LIN {X 0,Y 336.702,Z 407.414,A -85,B 0,C 180,E1 14263.606,E2 14263.606} C_VEL
LIN {X 0,Y 350.365,Z 438.947,A -85,B 0,C 180,E1 14267.093,E2 14267.093} C_VEL
LIN {X 0,Y 354.016,Z 453.085,A -85,B 0,C 180,E1 14268.481,E2 14268.481} C_VEL
LIN {X 0,Y 347.753,Z 489.705,A -85,B 0,C 180,E1 14270.853,E2 14270.853} C_VEL
LIN {X 0,Y 340.451,Z 523.229,A -85,B 0,C 180,E1 14274.153,E2 14274.153} C_VEL
LIN {X 0,Y 333.138,Z 552.708,A -85,B 0,C 180,E1 14278.297,E2 14278.297} C_VEL
LIN {X 0,Y 326.374,Z 579.149,A -85,B 0,C 180,E1 14283.478,E2 14283.478} C_VEL
LIN {X 0,Y 321.559,Z 600.193,A -85,B 0,C 180,E1 14289.32,E2 14289.32} C_VEL
LIN {X 0,Y 319.066,Z 615.775,A -85,B 0,C 180,E1 14295.571,E2 14295.571} C_VEL
LIN {X 0,Y 318.287,Z 625.498,A -85,B 0,C 180,E1 14301.792,E2 14301.792} C_VEL
LIN {X 0,Y 318.177,Z 629.765,A -85,B 0,C 180,E1 14307.742,E2 14307.742} C_VEL
LIN {X 0,Y 318.198,Z 629.579,A -85,B 0,C 180,E1 14312.723,E2 14312.723} C_VEL
LIN {X 0,Y 318.284,Z 625.522,A -85,B 0,C 180,E1 14318.2,E2 14318.2} C_VEL
LIN {X 0,Y 319.076,Z 615.81,A -85,B 0,C 180,E1 14324.42,E2 14324.42} C_VEL
LIN {X 0,Y 321.561,Z 600.254,A -85,B 0,C 180,E1 14330.672,E2 14330.672} C_VEL
LIN {X 0,Y 326.357,Z 579.231,A -85,B 0,C 180,E1 14336.514,E2 14336.514} C_VEL
LIN {X 0,Y 333.076,Z 552.834,A -85,B 0,C 180,E1 14341.701,E2 14341.701} C_VEL
LIN {X 0,Y 340.72,Z 522.288,A -85,B 0,C 180,E1 14345.973,E2 14345.973} C_VEL
LIN {X 0,Y 345.478,Z 500.812,A -85,B 0,C 180,E1 14348.213,E2 14348.213} C_VEL
LIN {X 0,Y 345.475,Z 486.2,A -85,B 0,C 180,E1 14349.823,E2 14349.823} C_VEL
LIN {X 0,Y 345.049,Z 471.082,A -85,B 0,C 180,E1 14351.299,E2 14351.299} C_VEL
LIN {X 0,Y 347.545,Z 452.345,A -85,B 0,C 180,E1 14352.445,E2 14352.445} C_VEL
LIN {X 0,Y 344.868,Z 441.835,A -85,B 0,C 180,E1 14353.735,E2 14353.735} C_VEL
LIN {X 0,Y 348.189,Z 426.338,A -85,B 0,C 180,E1 14356.65,E2 14356.65} C_VEL
LIN {X 0,Y 349.122,Z 427.681,A -85,B 0,C 180,E1 14358.678,E2 14358.678} C_VEL
LIN {X 0,Y 350.875,Z 436.55,A -85,B 0,C 180,E1 14361.396,E2 14361.396} C_VEL
LIN {X 0,Y 351.064,Z 446.749,A -85,B 0,C 180,E1 14362.964,E2 14362.964} C_VEL
LIN {X 0,Y 343.034,Z 479.923,A -85,B 0,C 180,E1 14365.756,E2 14365.756} C_VEL
LIN {X 0,Y 334.587,Z 510.275,A -85,B 0,C 180,E1 14369.506,E2 14369.506} C_VEL
LIN {X 0,Y 326.885,Z 535.038,A -85,B 0,C 180,E1 14373.896,E2 14373.896} C_VEL
LIN {X 0,Y 320.527,Z 554.48,A -85,B 0,C 180,E1 14378.889,E2 14378.889} C_VEL
LIN {X 0,Y 315.355,Z 569.315,A -85,B 0,C 180,E1 14384.689,E2 14384.689} C_VEL
LIN {X 0,Y 312.635,Z 577.44,A -85,B 0,C 180,E1 14390.24,E2 14390.24} C_VEL
LIN {X 0,Y 311.591,Z 580.289,A -85,B 0,C 180,E1 14394.422,E2 14394.422} C_VEL
LIN {X 0,Y 310.959,Z 579.837,A -85,B 0,C 180,E1 14399.998,E2 14399.998} C_VEL
LIN {X 0,Y 310.936,Z 574.542,A -85,B 0,C 180,E1 14405.586,E2 14405.586} C_VEL
LIN {X 0,Y 311.837,Z 563.945,A -85,B 0,C 180,E1 14411.196,E2 14411.196} C_VEL
LIN {X 0,Y 313.821,Z 548.299,A -85,B 0,C 180,E1 14416.516,E2 14416.516} C_VEL
LIN {X 0,Y 317.149,Z 526.048,A -85,B 0,C 180,E1 14421.701,E2 14421.701} C_VEL
LIN {X 0,Y 321.35,Z 498.61,A -85,B 0,C 180,E1 14426.18,E2 14426.18} C_VEL
LIN {X 0,Y 325.748,Z 466.866,A -85,B 0,C 180,E1 14429.78,E2 14429.78} C_VEL
LIN {X 0,Y 328.62,Z 434.304,A -85,B 0,C 180,E1 14432.319,E2 14432.319} C_VEL
LIN {X 0,Y 318.138,Z 399.395,A -85,B 0,C 180,E1 14434.97,E2 14434.97} C_VEL
LIN {X 0,Y 307.862,Z 370.16,A -85,B 0,C 180,E1 14437.035,E2 14437.035} C_VEL
LIN {X 0,Y 307.689,Z 370.824,A -85,B 0,C 180,E1 14441.794,E2 14441.794} C_VEL
LIN {X 0,Y 310.495,Z 376.206,A -85,B 0,C 180,E1 14442.604,E2 14442.604} C_VEL
LIN {X 0,Y 327.111,Z 403.706,A -85,B 0,C 180,E1 14446.915,E2 14446.915} C_VEL
LIN {X 0,Y 339.147,Z 431.187,A -85,B 0,C 180,E1 14450.634,E2 14450.634} C_VEL
LIN {X 0,Y 345.781,Z 455.325,A -85,B 0,C 180,E1 14453.75,E2 14453.75} C_VEL
LIN {X 0,Y 339.014,Z 485.871,A -85,B 0,C 180,E1 14456.649,E2 14456.649} C_VEL
LIN {X 0,Y 331.199,Z 513.667,A -85,B 0,C 180,E1 14460.534,E2 14460.534} C_VEL
LIN {X 0,Y 323.899,Z 536.369,A -85,B 0,C 180,E1 14465.128,E2 14465.128} C_VEL
LIN {X 0,Y 317.8,Z 554.685,A -85,B 0,C 180,E1 14470.525,E2 14470.525} C_VEL
LIN {X 0,Y 313.515,Z 568.434,A -85,B 0,C 180,E1 14476.744,E2 14476.744} C_VEL
LIN {X 0,Y 311.417,Z 576.322,A -85,B 0,C 180,E1 14483.023,E2 14483.023} C_VEL
LIN {X 0,Y 310.747,Z 579.252,A -85,B 0,C 180,E1 14490.004,E2 14490.004} C_VEL
LIN {X 0,Y 311.5,Z 576.22,A -85,B 0,C 180,E1 14496.983,E2 14496.983} C_VEL
LIN {X 0,Y 313.556,Z 568.228,A -85,B 0,C 180,E1 14503.263,E2 14503.263} C_VEL
LIN {X 0,Y 317.899,Z 554.376,A -85,B 0,C 180,E1 14509.477,E2 14509.477} C_VEL
LIN {X 0,Y 324.005,Z 535.911,A -85,B 0,C 180,E1 14514.872,E2 14514.872} C_VEL
LIN {X 0,Y 331.256,Z 513.253,A -85,B 0,C 180,E1 14519.431,E2 14519.431} C_VEL
LIN {X 0,Y 338.817,Z 486.357,A -85,B 0,C 180,E1 14523.191,E2 14523.191} C_VEL
LIN {X 0,Y 345.654,Z 455.489,A -85,B 0,C 180,E1 14526.133,E2 14526.133} C_VEL
LIN {X 0,Y 338.41,Z 429.395,A -85,B 0,C 180,E1 14529.496,E2 14529.496} C_VEL
LIN {X 0,Y 325.995,Z 401.987,A -85,B 0,C 180,E1 14533.24,E2 14533.24} C_VEL
LIN {X 0,Y 310.323,Z 376.076,A -85,B 0,C 180,E1 14537.302,E2 14537.302} C_VEL
LIN {X 0,Y 307.651,Z 370.931,A -85,B 0,C 180,E1 14538.072,E2 14538.072} C_VEL
LIN {X 0,Y 307.576,Z 370.16,A -85,B 0,C 180,E1 14543.799,E2 14543.799} C_VEL
LIN {X 0,Y 307.908,Z 370.16,A -85,B 0,C 180,E1 14552.264,E2 14552.264} C_VEL
LIN {X 0,Y 308.382,Z 370.16,A -85,B 0,C 180,E1 14559.903,E2 14559.903} C_VEL
LIN {X 0,Y 308.786,Z 370.16,A -85,B 0,C 180,E1 14565.812,E2 14565.812} C_VEL
LIN {X 0,Y 309.337,Z 370.16,A -85,B 0,C 180,E1 14574.385,E2 14574.385} C_VEL
LIN {X 0,Y 309.766,Z 370.16,A -85,B 0,C 180,E1 14580.002,E2 14580.002} C_VEL
LIN {X 0,Y 309.296,Z 370.16,A -85,B 0,C 180,E1 14585.62,E2 14585.62} C_VEL
LIN {X 0,Y 308.66,Z 370.16,A -85,B 0,C 180,E1 14594.198,E2 14594.198} C_VEL
LIN {X 0,Y 308.244,Z 370.16,A -85,B 0,C 180,E1 14601.053,E2 14601.053} C_VEL
LIN {X 0,Y 307.895,Z 370.16,A -85,B 0,C 180,E1 14609.454,E2 14609.454} C_VEL
LIN {X 0,Y 307.761,Z 370.16,A -85,B 0,C 180,E1 14616.747,E2 14616.747} C_VEL
LIN {X 0,Y 309.937,Z 375.586,A -85,B 0,C 180,E1 14617.459,E2 14617.459} C_VEL
LIN {X 0,Y 325.382,Z 400.525,A -85,B 0,C 180,E1 14621.422,E2 14621.422} C_VEL
LIN {X 0,Y 340.189,Z 430.993,A -85,B 0,C 180,E1 14625.193,E2 14625.193} C_VEL
LIN {X 0,Y 347.622,Z 453.192,A -85,B 0,C 180,E1 14627.648,E2 14627.648} C_VEL
LIN {X 0,Y 341.562,Z 488.7,A -85,B 0,C 180,E1 14630.002,E2 14630.002} C_VEL
LIN {X 0,Y 333.796,Z 522.751,A -85,B 0,C 180,E1 14633.38,E2 14633.38} C_VEL
LIN {X 0,Y 326.48,Z 550.936,A -85,B 0,C 180,E1 14637.375,E2 14637.375} C_VEL
LIN {X 0,Y 319.489,Z 576.93,A -85,B 0,C 180,E1 14642.478,E2 14642.478} C_VEL
LIN {X 0,Y 314.229,Z 598.464,A -85,B 0,C 180,E1 14648.442,E2 14648.442} C_VEL
LIN {X 0,Y 311.459,Z 613.662,A -85,B 0,C 180,E1 14654.49,E2 14654.49} C_VEL
LIN {X 0,Y 310.496,Z 623.14,A -85,B 0,C 180,E1 14660.17,E2 14660.17} C_VEL
LIN {X 0,Y 310.347,Z 627.396,A -85,B 0,C 180,E1 14664.397,E2 14664.397} C_VEL
LIN {X 0,Y 310.449,Z 629.513,A -85,B 0,C 180,E1 14669.996,E2 14669.996} C_VEL
LIN {X 0,Y 310.342,Z 627.41,A -85,B 0,C 180,E1 14675.595,E2 14675.595} C_VEL
LIN {X 0,Y 310.802,Z 619.779,A -85,B 0,C 180,E1 14682.194,E2 14682.194} C_VEL
LIN {X 0,Y 312.461,Z 607.513,A -85,B 0,C 180,E1 14688.272,E2 14688.272} C_VEL
LIN {X 0,Y 316.263,Z 589.869,A -85,B 0,C 180,E1 14694.207,E2 14694.207} C_VEL
LIN {X 0,Y 322.526,Z 565.801,A -85,B 0,C 180,E1 14699.927,E2 14699.927} C_VEL
LIN {X 0,Y 330.097,Z 537.476,A -85,B 0,C 180,E1 14704.714,E2 14704.714} C_VEL
LIN {X 0,Y 337.79,Z 505.842,A -85,B 0,C 180,E1 14708.484,E2 14708.484} C_VEL
LIN {X 0,Y 345.049,Z 471.082,A -85,B 0,C 180,E1 14711.299,E2 14711.299} C_VEL
LIN {X 0,Y 344.5,Z 459.969,A -85,B 0,C 180,E1 14712.439,E2 14712.439} C_VEL
LIN {X 0,Y 342.454,Z 446.059,A -85,B 0,C 180,E1 14714.842,E2 14714.842} C_VEL
LIN {X 0,Y 342.769,Z 444.544,A -85,B 0,C 180,E1 14715.112,E2 14715.112} C_VEL
LIN {X 0,Y 346.11,Z 433.791,A -85,B 0,C 180,E1 14717.188,E2 14717.188} C_VEL
LIN {X 0,Y 346.669,Z 436.725,A -85,B 0,C 180,E1 14719.074,E2 14719.074} C_VEL
LIN {X 0,Y 347.37,Z 443.98,A -85,B 0,C 180,E1 14721.068,E2 14721.068} C_VEL
LIN {X 0,Y 346.798,Z 450.589,A -85,B 0,C 180,E1 14722.008,E2 14722.008} C_VEL
LIN {X 0,Y 337.748,Z 483.682,A -85,B 0,C 180,E1 14724.947,E2 14724.947} C_VEL
LIN {X 0,Y 328.379,Z 513.691,A -85,B 0,C 180,E1 14728.866,E2 14728.866} C_VEL
LIN {X 0,Y 319.633,Z 538.965,A -85,B 0,C 180,E1 14733.636,E2 14733.636} C_VEL
LIN {X 0,Y 313.003,Z 557.38,A -85,B 0,C 180,E1 14738.729,E2 14738.729} C_VEL
LIN {X 0,Y 307.762,Z 570.989,A -85,B 0,C 180,E1 14744.45,E2 14744.45} C_VEL
LIN {X 0,Y 304.913,Z 578.511,A -85,B 0,C 180,E1 14749.991,E2 14749.991} C_VEL
LIN {X 0,Y 303.429,Z 581.458,A -85,B 0,C 180,E1 14756.204,E2 14756.204} C_VEL
LIN {X 0,Y 302.89,Z 579.333,A -85,B 0,C 180,E1 14761.659,E2 14761.659} C_VEL
LIN {X 0,Y 303.226,Z 572.681,A -85,B 0,C 180,E1 14767.168,E2 14767.168} C_VEL
LIN {X 0,Y 304.477,Z 560.301,A -85,B 0,C 180,E1 14772.927,E2 14772.927} C_VEL
LIN {X 0,Y 306.94,Z 542.722,A -85,B 0,C 180,E1 14778.325,E2 14778.325} C_VEL
LIN {X 0,Y 310.489,Z 519.357,A -85,B 0,C 180,E1 14783.337,E2 14783.337} C_VEL
LIN {X 0,Y 314.973,Z 490.822,A -85,B 0,C 180,E1 14787.639,E2 14787.639} C_VEL
LIN {X 0,Y 319.406,Z 458.406,A -85,B 0,C 180,E1 14791.025,E2 14791.025} C_VEL
LIN {X 0,Y 321.244,Z 436.106,A -85,B 0,C 180,E1 14792.722,E2 14792.722} C_VEL
LIN {X 0,Y 310.662,Z 400.803,A -85,B 0,C 180,E1 14795.523,E2 14795.523} C_VEL
LIN {X 0,Y 299.853,Z 370.16,A -85,B 0,C 180,E1 14797.745,E2 14797.745} C_VEL
LIN {X 0,Y 299.74,Z 370.16,A -85,B 0,C 180,E1 14799.872,E2 14799.872} C_VEL
LIN {X 0,Y 301.856,Z 375.542,A -85,B 0,C 180,E1 14800.591,E2 14800.591} C_VEL
LIN {X 0,Y 315.498,Z 396.485,A -85,B 0,C 180,E1 14804.365,E2 14804.365} C_VEL
LIN {X 0,Y 329.289,Z 424.408,A -85,B 0,C 180,E1 14808.534,E2 14808.534} C_VEL
LIN {X 0,Y 338.307,Z 452.752,A -85,B 0,C 180,E1 14812.426,E2 14812.426} C_VEL
LIN {X 0,Y 338.942,Z 459.143,A -85,B 0,C 180,E1 14813.205,E2 14813.205} C_VEL
LIN {X 0,Y 331.781,Z 489.358,A -85,B 0,C 180,E1 14816.217,E2 14816.217} C_VEL
LIN {X 0,Y 323.765,Z 516.226,A -85,B 0,C 180,E1 14820.171,E2 14820.171} C_VEL
LIN {X 0,Y 316.084,Z 538.932,A -85,B 0,C 180,E1 14824.995,E2 14824.995} C_VEL
LIN {X 0,Y 309.689,Z 557.189,A -85,B 0,C 180,E1 14830.737,E2 14830.737} C_VEL
LIN {X 0,Y 305.478,Z 570.202,A -85,B 0,C 180,E1 14837.118,E2 14837.118} C_VEL
LIN {X 0,Y 303.583,Z 576.961,A -85,B 0,C 180,E1 14842.842,E2 14842.842} C_VEL
LIN {X 0,Y 302.872,Z 579.889,A -85,B 0,C 180,E1 14850.004,E2 14850.004} C_VEL
LIN {X 0,Y 303.681,Z 576.859,A -85,B 0,C 180,E1 14857.164,E2 14857.164} C_VEL
LIN {X 0,Y 305.854,Z 568.877,A -85,B 0,C 180,E1 14863.603,E2 14863.603} C_VEL
LIN {X 0,Y 310.459,Z 555.034,A -85,B 0,C 180,E1 14869.964,E2 14869.964} C_VEL
LIN {X 0,Y 316.849,Z 536.599,A -85,B 0,C 180,E1 14875.474,E2 14875.474} C_VEL
LIN {X 0,Y 324.501,Z 513.743,A -85,B 0,C 180,E1 14880.154,E2 14880.154} C_VEL
LIN {X 0,Y 332.652,Z 485.813,A -85,B 0,C 180,E1 14884.085,E2 14884.085} C_VEL
LIN {X 0,Y 338.965,Z 455.987,A -85,B 0,C 180,E1 14887.02,E2 14887.02} C_VEL
LIN {X 0,Y 330.607,Z 428.038,A -85,B 0,C 180,E1 14890.858,E2 14890.858} C_VEL
LIN {X 0,Y 317.076,Z 399.156,A -85,B 0,C 180,E1 14895.071,E2 14895.071} C_VEL
LIN {X 0,Y 302.296,Z 376.02,A -85,B 0,C 180,E1 14899.145,E2 14899.145} C_VEL
LIN {X 0,Y 299.843,Z 371.763,A -85,B 0,C 180,E1 14899.898,E2 14899.898} C_VEL
LIN {X 0,Y 299.713,Z 370.16,A -85,B 0,C 180,E1 14900.105,E2 14900.105} C_VEL
LIN {X 0,Y 299.69,Z 370.16,A -85,B 0,C 180,E1 14906.245,E2 14906.245} C_VEL
LIN {X 0,Y 300.052,Z 370.16,A -85,B 0,C 180,E1 14912.996,E2 14912.996} C_VEL
LIN {X 0,Y 300.411,Z 370.16,A -85,B 0,C 180,E1 14919.346,E2 14919.346} C_VEL
LIN {X 0,Y 300.816,Z 370.16,A -85,B 0,C 180,E1 14925.428,E2 14925.428} C_VEL
LIN {X 0,Y 301.406,Z 370.16,A -85,B 0,C 180,E1 14934.236,E2 14934.236} C_VEL
LIN {X 0,Y 301.876,Z 370.16,A -85,B 0,C 180,E1 14940.002,E2 14940.002} C_VEL
LIN {X 0,Y 301.369,Z 370.16,A -85,B 0,C 180,E1 14945.768,E2 14945.768} C_VEL
LIN {X 0,Y 300.697,Z 370.16,A -85,B 0,C 180,E1 14954.582,E2 14954.582} C_VEL
LIN {X 0,Y 300.386,Z 370.16,A -85,B 0,C 180,E1 14960.66,E2 14960.66} C_VEL
LIN {X 0,Y 300.06,Z 370.16,A -85,B 0,C 180,E1 14967.008,E2 14967.008} C_VEL
LIN {X 0,Y 299.719,Z 370.5,A -85,B 0,C 180,E1 14974.873,E2 14974.873} C_VEL
LIN {X 0,Y 302.327,Z 375.981,A -85,B 0,C 180,E1 14975.728,E2 14975.728} C_VEL
LIN {X 0,Y 317.853,Z 400.489,A -85,B 0,C 180,E1 14979.998,E2 14979.998} C_VEL
LIN {X 0,Y 332.471,Z 429.96,A -85,B 0,C 180,E1 14983.926,E2 14983.926} C_VEL
LIN {X 0,Y 341.093,Z 455.224,A -85,B 0,C 180,E1 14986.899,E2 14986.899} C_VEL
LIN {X 0,Y 334.605,Z 491.504,A -85,B 0,C 180,E1 14989.423,E2 14989.423} C_VEL
LIN {X 0,Y 326.491,Z 525.053,A -85,B 0,C 180,E1 14992.924,E2 14992.924} C_VEL
LIN {X 0,Y 318.547,Z 554.163,A -85,B 0,C 180,E1 14997.27,E2 14997.27} C_VEL
LIN {X 0,Y 311.072,Z 580.518,A -85,B 0,C 180,E1 15002.849,E2 15002.849} C_VEL
LIN {X 0,Y 305.934,Z 600.89,A -85,B 0,C 180,E1 15008.971,E2 15008.971} C_VEL
LIN {X 0,Y 303.271,Z 615.82,A -85,B 0,C 180,E1 15015.542,E2 15015.542} C_VEL
LIN {X 0,Y 302.512,Z 624.197,A -85,B 0,C 180,E1 15021.361,E2 15021.361} C_VEL
LIN {X 0,Y 302.434,Z 628.293,A -85,B 0,C 180,E1 15027.126,E2 15027.126} C_VEL
LIN {X 0,Y 302.433,Z 628.302,A -85,B 0,C 180,E1 15032.865,E2 15032.865} C_VEL
LIN {X 0,Y 302.512,Z 624.223,A -85,B 0,C 180,E1 15038.63,E2 15038.63} C_VEL
LIN {X 0,Y 303.498,Z 614.481,A -85,B 0,C 180,E1 15045.177,E2 15045.177} C_VEL
LIN {X 0,Y 306.449,Z 598.884,A -85,B 0,C 180,E1 15051.743,E2 15051.743} C_VEL
LIN {X 0,Y 311.857,Z 577.812,A -85,B 0,C 180,E1 15057.851,E2 15057.851} C_VEL
LIN {X 0,Y 319.012,Z 552.302,A -85,B 0,C 180,E1 15063.071,E2 15063.071} C_VEL
LIN {X 0,Y 327.418,Z 521.78,A -85,B 0,C 180,E1 15067.498,E2 15067.498} C_VEL
LIN {X 0,Y 335.044,Z 489.942,A -85,B 0,C 180,E1 15070.716,E2 15070.716} C_VEL
LIN {X 0,Y 341.106,Z 454.446,A -85,B 0,C 180,E1 15073.22,E2 15073.22} C_VEL
LIN {X 0,Y 342.769,Z 444.544,A -85,B 0,C 180,E1 15075.112,E2 15075.112} C_VEL
LIN {X 0,Y 343.678,Z 441.281,A -85,B 0,C 180,E1 15076.489,E2 15076.489} C_VEL
LIN {X 0,Y 343.81,Z 443.304,A -85,B 0,C 180,E1 15078.573,E2 15078.573} C_VEL
LIN {X 0,Y 343.839,Z 444.628,A -85,B 0,C 180,E1 15079.064,E2 15079.064} C_VEL
LIN {X 0,Y 343.379,Z 452.909,A -85,B 0,C 180,E1 15080.894,E2 15080.894} C_VEL
LIN {X 0,Y 333.025,Z 486.412,A -85,B 0,C 180,E1 15083.974,E2 15083.974} C_VEL
LIN {X 0,Y 322.316,Z 517.144,A -85,B 0,C 180,E1 15088.175,E2 15088.175} C_VEL
LIN {X 0,Y 312.971,Z 541.55,A -85,B 0,C 180,E1 15093.03,E2 15093.03} C_VEL
LIN {X 0,Y 305.882,Z 559.257,A -85,B 0,C 180,E1 15098.208,E2 15098.208} C_VEL
LIN {X 0,Y 300.292,Z 572.35,A -85,B 0,C 180,E1 15104.007,E2 15104.007} C_VEL
LIN {X 0,Y 297.197,Z 579.631,A -85,B 0,C 180,E1 15109.728,E2 15109.728} C_VEL
LIN {X 0,Y 295.954,Z 582.027,A -85,B 0,C 180,E1 15114.126,E2 15114.126} C_VEL
LIN {X 0,Y 295.216,Z 581.023,A -85,B 0,C 180,E1 15119.998,E2 15119.998} C_VEL
LIN {X 0,Y 295.189,Z 575.183,A -85,B 0,C 180,E1 15125.885,E2 15125.885} C_VEL
LIN {X 0,Y 296.227,Z 563.913,A -85,B 0,C 180,E1 15131.794,E2 15131.794} C_VEL
LIN {X 0,Y 298.61,Z 546.312,A -85,B 0,C 180,E1 15137.707,E2 15137.707} C_VEL
LIN {X 0,Y 302.263,Z 523.292,A -85,B 0,C 180,E1 15142.995,E2 15142.995} C_VEL
LIN {X 0,Y 306.656,Z 496.066,A -85,B 0,C 180,E1 15147.407,E2 15147.407} C_VEL
LIN {X 0,Y 311.404,Z 463.285,A -85,B 0,C 180,E1 15151.098,E2 15151.098} C_VEL
LIN {X 0,Y 313.631,Z 437.042,A -85,B 0,C 180,E1 15153.218,E2 15153.218} C_VEL
LIN {X 0,Y 303.454,Z 402.954,A -85,B 0,C 180,E1 15156.029,E2 15156.029} C_VEL
LIN {X 0,Y 292.915,Z 373.981,A -85,B 0,C 180,E1 15158.237,E2 15158.237} C_VEL
LIN {X 0,Y 300.967,Z 385.635,A -85,B 0,C 180,E1 15160.736,E2 15160.736} C_VEL
LIN {X 0,Y 315.245,Z 409.626,A -85,B 0,C 180,E1 15164.976,E2 15164.976} C_VEL
LIN {X 0,Y 326.932,Z 437.652,A -85,B 0,C 180,E1 15169.192,E2 15169.192} C_VEL
LIN {X 0,Y 332.617,Z 460.462,A -85,B 0,C 180,E1 15172.426,E2 15172.426} C_VEL
LIN {X 0,Y 324.893,Z 491.471,A -85,B 0,C 180,E1 15175.62,E2 15175.62} C_VEL
LIN {X 0,Y 316.388,Z 518.604,A -85,B 0,C 180,E1 15179.758,E2 15179.758} C_VEL
LIN {X 0,Y 308.526,Z 540.66,A -85,B 0,C 180,E1 15184.662,E2 15184.662} C_VEL
LIN {X 0,Y 302.237,Z 557.844,A -85,B 0,C 180,E1 15190.243,E2 15190.243} C_VEL
LIN {X 0,Y 297.777,Z 570.844,A -85,B 0,C 180,E1 15196.779,E2 15196.779} C_VEL
LIN {X 0,Y 295.752,Z 577.599,A -85,B 0,C 180,E1 15202.652,E2 15202.652} C_VEL
LIN {X 0,Y 294.997,Z 580.526,A -85,B 0,C 180,E1 15210.004,E2 15210.004} C_VEL
LIN {X 0,Y 295.847,Z 577.499,A -85,B 0,C 180,E1 15217.355,E2 15217.355} C_VEL
LIN {X 0,Y 298.189,Z 569.525,A -85,B 0,C 180,E1 15223.96,E2 15223.96} C_VEL
LIN {X 0,Y 303.031,Z 555.692,A -85,B 0,C 180,E1 15230.475,E2 15230.475} C_VEL
LIN {X 0,Y 309.734,Z 537.287,A -85,B 0,C 180,E1 15236.102,E2 15236.102} C_VEL
LIN {X 0,Y 317.996,Z 513.573,A -85,B 0,C 180,E1 15241.029,E2 15241.029} C_VEL
LIN {X 0,Y 326.166,Z 486.631,A -85,B 0,C 180,E1 15244.859,E2 15244.859} C_VEL
LIN {X 0,Y 332.37,Z 458.432,A -85,B 0,C 180,E1 15247.72,E2 15247.72} C_VEL
LIN {X 0,Y 324.821,Z 431.908,A -85,B 0,C 180,E1 15251.527,E2 15251.527} C_VEL
LIN {X 0,Y 312.463,Z 404.48,A -85,B 0,C 180,E1 15255.736,E2 15255.736} C_VEL
LIN {X 0,Y 298.461,Z 382.046,A -85,B 0,C 180,E1 15259.865,E2 15259.865} C_VEL
LIN {X 0,Y 293.925,Z 375.589,A -85,B 0,C 180,E1 15261.277,E2 15261.277} C_VEL
LIN {X 0,Y 291.724,Z 370.16,A -85,B 0,C 180,E1 15262.142,E2 15262.142} C_VEL
LIN {X 0,Y 291.852,Z 370.16,A -85,B 0,C 180,E1 15268.756,E2 15268.756} C_VEL
LIN {X 0,Y 292.214,Z 370.16,A -85,B 0,C 180,E1 15275.517,E2 15275.517} C_VEL
LIN {X 0,Y 292.639,Z 370.16,A -85,B 0,C 180,E1 15281.919,E2 15281.919} C_VEL
LIN {X 0,Y 293.076,Z 370.16,A -85,B 0,C 180,E1 15288.977,E2 15288.977} C_VEL
LIN {X 0,Y 293.734,Z 370.16,A -85,B 0,C 180,E1 15297.048,E2 15297.048} C_VEL
LIN {X 0,Y 293.762,Z 370.16,A -85,B 0,C 180,E1 15302.956,E2 15302.956} C_VEL
LIN {X 0,Y 292.98,Z 370.16,A -85,B 0,C 180,E1 15311.93,E2 15311.93} C_VEL
LIN {X 0,Y 292.567,Z 370.16,A -85,B 0,C 180,E1 15318.09,E2 15318.09} C_VEL
LIN {X 0,Y 292.213,Z 370.16,A -85,B 0,C 180,E1 15324.488,E2 15324.488} C_VEL
LIN {X 0,Y 291.8,Z 370.16,A -85,B 0,C 180,E1 15332.753,E2 15332.753} C_VEL
LIN {X 0,Y 294.044,Z 375.638,A -85,B 0,C 180,E1 15333.625,E2 15333.625} C_VEL
LIN {X 0,Y 307.27,Z 395.323,A -85,B 0,C 180,E1 15337.611,E2 15337.611} C_VEL
LIN {X 0,Y 323.041,Z 424.864,A -85,B 0,C 180,E1 15342.033,E2 15342.033} C_VEL
LIN {X 0,Y 333.881,Z 454.652,A -85,B 0,C 180,E1 15345.808,E2 15345.808} C_VEL
LIN {X 0,Y 334.19,Z 462.513,A -85,B 0,C 180,E1 15346.497,E2 15346.497} C_VEL
LIN {X 0,Y 326.862,Z 497.513,A -85,B 0,C 180,E1 15349.134,E2 15349.134} C_VEL
LIN {X 0,Y 318.284,Z 530.567,A -85,B 0,C 180,E1 15352.875,E2 15352.875} C_VEL
LIN {X 0,Y 310.02,Z 558.973,A -85,B 0,C 180,E1 15357.504,E2 15357.504} C_VEL
LIN {X 0,Y 302.685,Z 583.975,A -85,B 0,C 180,E1 15363.242,E2 15363.242} C_VEL
LIN {X 0,Y 297.628,Z 603.487,A -85,B 0,C 180,E1 15369.683,E2 15369.683} C_VEL
LIN {X 0,Y 295.234,Z 617.007,A -85,B 0,C 180,E1 15376.262,E2 15376.262} C_VEL
LIN {X 0,Y 294.593,Z 624.934,A -85,B 0,C 180,E1 15382.614,E2 15382.614} C_VEL
LIN {X 0,Y 294.546,Z 627.653,A -85,B 0,C 180,E1 15387.049,E2 15387.049} C_VEL
LIN {X 0,Y 294.545,Z 627.662,A -85,B 0,C 180,E1 15392.942,E2 15392.942} C_VEL
LIN {X 0,Y 294.629,Z 623.574,A -85,B 0,C 180,E1 15398.863,E2 15398.863} C_VEL
LIN {X 0,Y 295.726,Z 613.817,A -85,B 0,C 180,E1 15405.586,E2 15405.586} C_VEL
LIN {X 0,Y 298.91,Z 598.2,A -85,B 0,C 180,E1 15412.321,E2 15412.321} C_VEL
LIN {X 0,Y 304.711,Z 577.107,A -85,B 0,C 180,E1 15418.564,E2 15418.564} C_VEL
LIN {X 0,Y 312.508,Z 550.528,A -85,B 0,C 180,E1 15424.064,E2 15424.064} C_VEL
LIN {X 0,Y 321.272,Z 519.948,A -85,B 0,C 180,E1 15428.51,E2 15428.51} C_VEL
LIN {X 0,Y 329.376,Z 487.046,A -85,B 0,C 180,E1 15431.79,E2 15431.79} C_VEL
LIN {X 0,Y 338.071,Z 458.881,A -85,B 0,C 180,E1 15434.232,E2 15434.232} C_VEL
LIN {X 0,Y 343.688,Z 441.716,A -85,B 0,C 180,E1 15437.626,E2 15437.626} C_VEL
LIN {X 0,Y 343.839,Z 444.628,A -85,B 0,C 180,E1 15439.064,E2 15439.064} C_VEL
LIN {X 0,Y 342.791,Z 449.901,A -85,B 0,C 180,E1 15439.817,E2 15439.817} C_VEL
LIN {X 0,Y 337.052,Z 465.549,A -85,B 0,C 180,E1 15440.55,E2 15440.55} C_VEL
LIN {X 0,Y 325.338,Z 497.939,A -85,B 0,C 180,E1 15444.019,E2 15444.019} C_VEL
LIN {X 0,Y 314.21,Z 525.939,A -85,B 0,C 180,E1 15448.399,E2 15448.399} C_VEL
LIN {X 0,Y 304.656,Z 548.119,A -85,B 0,C 180,E1 15453.432,E2 15453.432} C_VEL
LIN {X 0,Y 297.113,Z 564.887,A -85,B 0,C 180,E1 15459.102,E2 15459.102} C_VEL
LIN {X 0,Y 291.875,Z 575.89,A -85,B 0,C 180,E1 15464.967,E2 15464.967} C_VEL
LIN {X 0,Y 288.903,Z 581.759,A -85,B 0,C 180,E1 15470.953,E2 15470.953} C_VEL
LIN {X 0,Y 287.635,Z 582.871,A -85,B 0,C 180,E1 15476.981,E2 15476.981} C_VEL
LIN {X 0,Y 287.092,Z 579.127,A -85,B 0,C 180,E1 15483.021,E2 15483.021} C_VEL
LIN {X 0,Y 287.787,Z 570.371,A -85,B 0,C 180,E1 15489.078,E2 15489.078} C_VEL
LIN {X 0,Y 289.481,Z 555.69,A -85,B 0,C 180,E1 15495.156,E2 15495.156} C_VEL
LIN {X 0,Y 292.685,Z 535.296,A -85,B 0,C 180,E1 15500.829,E2 15500.829} C_VEL
LIN {X 0,Y 296.996,Z 509.359,A -85,B 0,C 180,E1 15505.876,E2 15505.876} C_VEL
LIN {X 0,Y 301.657,Z 479.435,A -85,B 0,C 180,E1 15509.967,E2 15509.967} C_VEL
LIN {X 0,Y 306.284,Z 444.892,A -85,B 0,C 180,E1 15513.172,E2 15513.172} C_VEL
LIN {X 0,Y 305.56,Z 436.302,A -85,B 0,C 180,E1 15513.9,E2 15513.9} C_VEL
LIN {X 0,Y 295.039,Z 401.661,A -85,B 0,C 180,E1 15516.807,E2 15516.807} C_VEL
LIN {X 0,Y 290.089,Z 387.094,A -85,B 0,C 180,E1 15517.979,E2 15517.979} C_VEL
LIN {X 0,Y 294.023,Z 386.917,A -85,B 0,C 180,E1 15519.034,E2 15519.034} C_VEL
LIN {X 0,Y 307.712,Z 409.353,A -85,B 0,C 180,E1 15523.39,E2 15523.39} C_VEL
LIN {X 0,Y 319.43,Z 436.496,A -85,B 0,C 180,E1 15527.776,E2 15527.776} C_VEL
LIN {X 0,Y 326.228,Z 461.91,A -85,B 0,C 180,E1 15531.613,E2 15531.613} C_VEL
LIN {X 0,Y 318.441,Z 492.257,A -85,B 0,C 180,E1 15534.823,E2 15534.823} C_VEL
LIN {X 0,Y 309.812,Z 518.675,A -85,B 0,C 180,E1 15538.904,E2 15538.904} C_VEL
LIN {X 0,Y 301.489,Z 541.123,A -85,B 0,C 180,E1 15543.962,E2 15543.962} C_VEL
LIN {X 0,Y 294.784,Z 558.5,A -85,B 0,C 180,E1 15549.721,E2 15549.721} C_VEL
LIN {X 0,Y 290.088,Z 571.486,A -85,B 0,C 180,E1 15556.422,E2 15556.422} C_VEL
LIN {X 0,Y 287.948,Z 578.236,A -85,B 0,C 180,E1 15562.452,E2 15562.452} C_VEL
LIN {X 0,Y 287.14,Z 581.162,A -85,B 0,C 180,E1 15570.005,E2 15570.005} C_VEL
LIN {X 0,Y 288.027,Z 578.138,A -85,B 0,C 180,E1 15577.555,E2 15577.555} C_VEL
LIN {X 0,Y 290.525,Z 570.172,A -85,B 0,C 180,E1 15584.336,E2 15584.336} C_VEL
LIN {X 0,Y 295.629,Z 556.349,A -85,B 0,C 180,E1 15591.011,E2 15591.011} C_VEL
LIN {X 0,Y 302.667,Z 537.97,A -85,B 0,C 180,E1 15596.76,E2 15596.76} C_VEL
LIN {X 0,Y 311.008,Z 515.044,A -85,B 0,C 180,E1 15601.641,E2 15601.641} C_VEL
LIN {X 0,Y 319.754,Z 487.449,A -85,B 0,C 180,E1 15605.664,E2 15605.664} C_VEL
LIN {X 0,Y 326.032,Z 461.717,A -85,B 0,C 180,E1 15608.317,E2 15608.317} C_VEL
LIN {X 0,Y 318.919,Z 435.361,A -85,B 0,C 180,E1 15612.285,E2 15612.285} C_VEL
LIN {X 0,Y 306.98,Z 408.176,A -85,B 0,C 180,E1 15616.704,E2 15616.704} C_VEL
LIN {X 0,Y 294.242,Z 387.325,A -85,B 0,C 180,E1 15620.743,E2 15620.743} C_VEL
LIN {X 0,Y 286.806,Z 376.351,A -85,B 0,C 180,E1 15623.24,E2 15623.24} C_VEL
LIN {X 0,Y 283.948,Z 371.74,A -85,B 0,C 180,E1 15624.297,E2 15624.297} C_VEL
LIN {X 0,Y 283.803,Z 370.16,A -85,B 0,C 180,E1 15624.611,E2 15624.611} C_VEL
LIN {X 0,Y 284.008,Z 370.16,A -85,B 0,C 180,E1 15631.334,E2 15631.334} C_VEL
LIN {X 0,Y 284.393,Z 370.16,A -85,B 0,C 180,E1 15638.124,E2 15638.124} C_VEL
LIN {X 0,Y 284.893,Z 370.16,A -85,B 0,C 180,E1 15644.594,E2 15644.594} C_VEL
LIN {X 0,Y 285.258,Z 370.16,A -85,B 0,C 180,E1 15651.474,E2 15651.474} C_VEL
LIN {X 0,Y 286.069,Z 370.16,A -85,B 0,C 180,E1 15660.002,E2 15660.002} C_VEL
LIN {X 0,Y 285.493,Z 370.16,A -85,B 0,C 180,E1 15666.09,E2 15666.09} C_VEL
LIN {X 0,Y 285.013,Z 370.16,A -85,B 0,C 180,E1 15672.269,E2 15672.269} C_VEL
LIN {X 0,Y 284.603,Z 370.16,A -85,B 0,C 180,E1 15678.614,E2 15678.614} C_VEL
LIN {X 0,Y 284.196,Z 370.16,A -85,B 0,C 180,E1 15685.226,E2 15685.226} C_VEL
LIN {X 0,Y 283.951,Z 370.16,A -85,B 0,C 180,E1 15690.433,E2 15690.433} C_VEL
LIN {X 0,Y 286.359,Z 375.83,A -85,B 0,C 180,E1 15691.481,E2 15691.481} C_VEL
LIN {X 0,Y 289.281,Z 380.069,A -85,B 0,C 180,E1 15692.513,E2 15692.513} C_VEL
LIN {X 0,Y 303.476,Z 401.499,A -85,B 0,C 180,E1 15696.995,E2 15696.995} C_VEL
LIN {X 0,Y 317.755,Z 429.287,A -85,B 0,C 180,E1 15701.334,E2 15701.334} C_VEL
LIN {X 0,Y 327.823,Z 458.123,A -85,B 0,C 180,E1 15705.156,E2 15705.156} C_VEL
LIN {X 0,Y 327.865,Z 464.079,A -85,B 0,C 180,E1 15705.696,E2 15705.696} C_VEL
LIN {X 0,Y 319.95,Z 500.034,A -85,B 0,C 180,E1 15708.508,E2 15708.508} C_VEL
LIN {X 0,Y 311.138,Z 532.144,A -85,B 0,C 180,E1 15712.314,E2 15712.314} C_VEL
LIN {X 0,Y 302.616,Z 560.037,A -85,B 0,C 180,E1 15717.031,E2 15717.031} C_VEL
LIN {X 0,Y 294.99,Z 584.6,A -85,B 0,C 180,E1 15722.917,E2 15722.917} C_VEL
LIN {X 0,Y 289.753,Z 603.898,A -85,B 0,C 180,E1 15729.575,E2 15729.575} C_VEL
LIN {X 0,Y 287.231,Z 617.755,A -85,B 0,C 180,E1 15736.763,E2 15736.763} C_VEL
LIN {X 0,Y 286.701,Z 625.469,A -85,B 0,C 180,E1 15743.933,E2 15743.933} C_VEL
LIN {X 0,Y 286.815,Z 627.601,A -85,B 0,C 180,E1 15749.995,E2 15749.995} C_VEL
LIN {X 0,Y 286.695,Z 625.485,A -85,B 0,C 180,E1 15756.058,E2 15756.058} C_VEL
LIN {X 0,Y 287.265,Z 617.738,A -85,B 0,C 180,E1 15763.262,E2 15763.262} C_VEL
LIN {X 0,Y 289.732,Z 603.962,A -85,B 0,C 180,E1 15770.416,E2 15770.416} C_VEL
LIN {X 0,Y 294.48,Z 586.044,A -85,B 0,C 180,E1 15776.681,E2 15776.681} C_VEL
LIN {X 0,Y 302.064,Z 561.927,A -85,B 0,C 180,E1 15782.614,E2 15782.614} C_VEL
LIN {X 0,Y 310.853,Z 533.533,A -85,B 0,C 180,E1 15787.496,E2 15787.496} C_VEL
LIN {X 0,Y 324.243,Z 492.274,A -85,B 0,C 180,E1 15792.606,E2 15792.606} C_VEL
LIN {X 0,Y 335.347,Z 463.531,A -85,B 0,C 180,E1 15795.241,E2 15795.241} C_VEL
LIN {X 0,Y 339.978,Z 451.725,A -85,B 0,C 180,E1 15797.628,E2 15797.628} C_VEL
LIN {X 0,Y 340.841,Z 450.441,A -85,B 0,C 180,E1 15798.219,E2 15798.219} C_VEL
LIN {X 0,Y 340.331,Z 455.505,A -85,B 0,C 180,E1 15799.688,E2 15799.688} C_VEL
LIN {X 0,Y 337.052,Z 465.549,A -85,B 0,C 180,E1 15800.55,E2 15800.55} C_VEL
LIN {X 0,Y 332.029,Z 476.365,A -85,B 0,C 180,E1 15800.831,E2 15800.831} C_VEL
LIN {X 0,Y 327.389,Z 485.432,A -85,B 0,C 180,E1 15801.094,E2 15801.094} C_VEL
LIN {X 0,Y 326.892,Z 486.611,A -85,B 0,C 180,E1 15801.213,E2 15801.213} C_VEL
LIN {X 0,Y 313.584,Z 517.523,A -85,B 0,C 180,E1 15805.484,E2 15805.484} C_VEL
LIN {X 0,Y 301.73,Z 543.01,A -85,B 0,C 180,E1 15810.71,E2 15810.71} C_VEL
LIN {X 0,Y 292.701,Z 561.435,A -85,B 0,C 180,E1 15816.367,E2 15816.367} C_VEL
LIN {X 0,Y 285.567,Z 574.969,A -85,B 0,C 180,E1 15822.901,E2 15822.901} C_VEL
LIN {X 0,Y 281.81,Z 581.908,A -85,B 0,C 180,E1 15829.161,E2 15829.161} C_VEL
LIN {X 0,Y 280.329,Z 583.744,A -85,B 0,C 180,E1 15833.797,E2 15833.797} C_VEL
LIN {X 0,Y 279.46,Z 582.172,A -85,B 0,C 180,E1 15839.998,E2 15839.998} C_VEL
LIN {X 0,Y 279.58,Z 574.455,A -85,B 0,C 180,E1 15846.996,E2 15846.996} C_VEL
LIN {X 0,Y 280.976,Z 561.211,A -85,B 0,C 180,E1 15853.443,E2 15853.443} C_VEL
LIN {X 0,Y 283.837,Z 542.208,A -85,B 0,C 180,E1 15859.471,E2 15859.471} C_VEL
LIN {X 0,Y 287.92,Z 517.629,A -85,B 0,C 180,E1 15864.873,E2 15864.873} C_VEL
LIN {X 0,Y 292.939,Z 488.157,A -85,B 0,C 180,E1 15869.401,E2 15869.401} C_VEL
LIN {X 0,Y 297.677,Z 455.038,A -85,B 0,C 180,E1 15872.906,E2 15872.906} C_VEL
LIN {X 0,Y 298.745,Z 440.346,A -85,B 0,C 180,E1 15874.11,E2 15874.11} C_VEL
LIN {X 0,Y 288.448,Z 405.504,A -85,B 0,C 180,E1 15877.221,E2 15877.221} C_VEL
LIN {X 0,Y 286.892,Z 400.24,A -85,B 0,C 180,E1 15877.702,E2 15877.702} C_VEL
LIN {X 0,Y 290.053,Z 399.029,A -85,B 0,C 180,E1 15878.514,E2 15878.514} C_VEL
LIN {X 0,Y 292.411,Z 395.613,A -85,B 0,C 180,E1 15878.988,E2 15878.988} C_VEL
LIN {X 0,Y 305.819,Z 420.407,A -85,B 0,C 180,E1 15883.746,E2 15883.746} C_VEL
LIN {X 0,Y 316.003,Z 448.066,A -85,B 0,C 180,E1 15888.308,E2 15888.308} C_VEL
LIN {X 0,Y 319.452,Z 466.064,A -85,B 0,C 180,E1 15891.042,E2 15891.042} C_VEL
LIN {X 0,Y 311.285,Z 495.391,A -85,B 0,C 180,E1 15894.3,E2 15894.3} C_VEL
LIN {X 0,Y 301.865,Z 522.679,A -85,B 0,C 180,E1 15898.779,E2 15898.779} C_VEL
LIN {X 0,Y 293.432,Z 544.267,A -85,B 0,C 180,E1 15903.994,E2 15903.994} C_VEL
LIN {X 0,Y 286.645,Z 560.933,A -85,B 0,C 180,E1 15909.927,E2 15909.927} C_VEL
LIN {X 0,Y 282.019,Z 573.204,A -85,B 0,C 180,E1 15916.817,E2 15916.817} C_VEL
LIN {X 0,Y 279.895,Z 579.954,A -85,B 0,C 180,E1 15923.794,E2 15923.794} C_VEL
LIN {X 0,Y 279.265,Z 581.799,A -85,B 0,C 180,E1 15930.005,E2 15930.005} C_VEL
LIN {X 0,Y 280.2,Z 578.778,A -85,B 0,C 180,E1 15937.768,E2 15937.768} C_VEL
LIN {X 0,Y 282.869,Z 570.82,A -85,B 0,C 180,E1 15944.732,E2 15944.732} C_VEL
LIN {X 0,Y 288.236,Z 557.007,A -85,B 0,C 180,E1 15951.577,E2 15951.577} C_VEL
LIN {X 0,Y 295.643,Z 538.654,A -85,B 0,C 180,E1 15957.448,E2 15957.448} C_VEL
LIN {X 0,Y 304.154,Z 516.259,A -85,B 0,C 180,E1 15962.327,E2 15962.327} C_VEL
LIN {X 0,Y 313.489,Z 487.993,A -85,B 0,C 180,E1 15966.533,E2 15966.533} C_VEL
LIN {X 0,Y 319.411,Z 463.27,A -85,B 0,C 180,E1 15969.199,E2 15969.199} C_VEL
LIN {X 0,Y 312.393,Z 436.859,A -85,B 0,C 180,E1 15973.374,E2 15973.374} C_VEL
LIN {X 0,Y 299.93,Z 408.667,A -85,B 0,C 180,E1 15978.271,E2 15978.271} C_VEL
LIN {X 0,Y 286.982,Z 387.883,A -85,B 0,C 180,E1 15982.71,E2 15982.71} C_VEL
LIN {X 0,Y 278.951,Z 376.352,A -85,B 0,C 180,E1 15985.689,E2 15985.689} C_VEL
LIN {X 0,Y 276.139,Z 371.699,A -85,B 0,C 180,E1 15986.873,E2 15986.873} C_VEL
LIN {X 0,Y 275.957,Z 370.16,A -85,B 0,C 180,E1 15987.197,E2 15987.197} C_VEL
LIN {X 0,Y 276.157,Z 370.16,A -85,B 0,C 180,E1 15993.99,E2 15993.99} C_VEL
LIN {X 0,Y 276.644,Z 370.16,A -85,B 0,C 180,E1 16000.834,E2 16000.834} C_VEL
LIN {X 0,Y 277.121,Z 370.16,A -85,B 0,C 180,E1 16007.38,E2 16007.38} C_VEL
LIN {X 0,Y 277.905,Z 370.16,A -85,B 0,C 180,E1 16016.879,E2 16016.879} C_VEL
LIN {X 0,Y 277.924,Z 370.16,A -85,B 0,C 180,E1 16023.125,E2 16023.125} C_VEL
LIN {X 0,Y 277.049,Z 370.16,A -85,B 0,C 180,E1 16032.628,E2 16032.628} C_VEL
LIN {X 0,Y 276.456,Z 370.16,A -85,B 0,C 180,E1 16041.403,E2 16041.403} C_VEL
LIN {X 0,Y 276.1,Z 370.546,A -85,B 0,C 180,E1 16047.914,E2 16047.914} C_VEL
LIN {X 0,Y 278.56,Z 375.9,A -85,B 0,C 180,E1 16049.033,E2 16049.033} C_VEL
LIN {X 0,Y 281.216,Z 379.311,A -85,B 0,C 180,E1 16050.069,E2 16050.069} C_VEL
LIN {X 0,Y 296.99,Z 403.168,A -85,B 0,C 180,E1 16055.527,E2 16055.527} C_VEL
LIN {X 0,Y 310.693,Z 429.449,A -85,B 0,C 180,E1 16059.987,E2 16059.987} C_VEL
LIN {X 0,Y 320.884,Z 458.307,A -85,B 0,C 180,E1 16064.056,E2 16064.056} C_VEL
LIN {X 0,Y 322.042,Z 463.637,A -85,B 0,C 180,E1 16064.744,E2 16064.744} C_VEL
LIN {X 0,Y 313.966,Z 499.112,A -85,B 0,C 180,E1 16067.535,E2 16067.535} C_VEL
LIN {X 0,Y 304.753,Z 531.345,A -85,B 0,C 180,E1 16071.381,E2 16071.381} C_VEL
LIN {X 0,Y 295.805,Z 559.311,A -85,B 0,C 180,E1 16076.175,E2 16076.175} C_VEL
LIN {X 0,Y 287.806,Z 583.681,A -85,B 0,C 180,E1 16082.11,E2 16082.11} C_VEL
LIN {X 0,Y 282.195,Z 602.946,A -85,B 0,C 180,E1 16088.882,E2 16088.882} C_VEL
LIN {X 0,Y 279.502,Z 616.331,A -85,B 0,C 180,E1 16095.889,E2 16095.889} C_VEL
LIN {X 0,Y 278.848,Z 623.643,A -85,B 0,C 180,E1 16102.194,E2 16102.194} C_VEL
LIN {X 0,Y 278.795,Z 626.376,A -85,B 0,C 180,E1 16106.883,E2 16106.883} C_VEL
LIN {X 0,Y 278.936,Z 626.963,A -85,B 0,C 180,E1 16109.995,E2 16109.995} C_VEL
LIN {X 0,Y 278.803,Z 624.842,A -85,B 0,C 180,E1 16116.23,E2 16116.23} C_VEL
LIN {X 0,Y 279.247,Z 618.462,A -85,B 0,C 180,E1 16122.608,E2 16122.608} C_VEL
LIN {X 0,Y 281.366,Z 606.542,A -85,B 0,C 180,E1 16129.528,E2 16129.528} C_VEL
LIN {X 0,Y 286.333,Z 588.345,A -85,B 0,C 180,E1 16136.502,E2 16136.502} C_VEL
LIN {X 0,Y 294.077,Z 564.629,A -85,B 0,C 180,E1 16142.716,E2 16142.716} C_VEL
LIN {X 0,Y 306.914,Z 527.619,A -85,B 0,C 180,E1 16149.421,E2 16149.421} C_VEL
LIN {X 0,Y 321.088,Z 494.632,A -85,B 0,C 180,E1 16153.824,E2 16153.824} C_VEL
LIN {X 0,Y 333.499,Z 466.711,A -85,B 0,C 180,E1 16156.574,E2 16156.574} C_VEL
LIN {X 0,Y 337.253,Z 459.12,A -85,B 0,C 180,E1 16158.138,E2 16158.138} C_VEL
LIN {X 0,Y 336.931,Z 460.946,A -85,B 0,C 180,E1 16158.781,E2 16158.781} C_VEL
LIN {X 0,Y 326.892,Z 486.611,A -85,B 0,C 180,E1 16161.213,E2 16161.213} C_VEL
LIN {X 0,Y 319.291,Z 501.337,A -85,B 0,C 180,E1 16162.299,E2 16162.299} C_VEL
LIN {X 0,Y 312.16,Z 513.499,A -85,B 0,C 180,E1 16163.343,E2 16163.343} C_VEL
LIN {X 0,Y 311.37,Z 515.045,A -85,B 0,C 180,E1 16163.578,E2 16163.578} C_VEL
LIN {X 0,Y 298.275,Z 540.698,A -85,B 0,C 180,E1 16168.649,E2 16168.649} C_VEL
LIN {X 0,Y 287.902,Z 559.852,A -85,B 0,C 180,E1 16174.288,E2 16174.288} C_VEL
LIN {X 0,Y 279.487,Z 574.434,A -85,B 0,C 180,E1 16181.032,E2 16181.032} C_VEL
LIN {X 0,Y 274.957,Z 581.868,A -85,B 0,C 180,E1 16187.275,E2 16187.275} C_VEL
LIN {X 0,Y 272.526,Z 584.617,A -85,B 0,C 180,E1 16193.619,E2 16193.619} C_VEL
LIN {X 0,Y 271.599,Z 582.66,A -85,B 0,C 180,E1 16199.998,E2 16199.998} C_VEL
LIN {X 0,Y 271.596,Z 575.784,A -85,B 0,C 180,E1 16206.399,E2 16206.399} C_VEL
LIN {X 0,Y 272.859,Z 563.395,A -85,B 0,C 180,E1 16212.82,E2 16212.82} C_VEL
LIN {X 0,Y 275.483,Z 545.811,A -85,B 0,C 180,E1 16218.834,E2 16218.834} C_VEL
LIN {X 0,Y 279.48,Z 522.433,A -85,B 0,C 180,E1 16224.393,E2 16224.393} C_VEL
LIN {X 0,Y 284.36,Z 494.521,A -85,B 0,C 180,E1 16229.063,E2 16229.063} C_VEL
LIN {X 0,Y 289.553,Z 461.255,A -85,B 0,C 180,E1 16232.911,E2 16232.911} C_VEL
LIN {X 0,Y 291.284,Z 442.018,A -85,B 0,C 180,E1 16234.574,E2 16234.574} C_VEL
LIN {X 0,Y 282.937,Z 412.441,A -85,B 0,C 180,E1 16237.405,E2 16237.405} C_VEL
LIN {X 0,Y 286.392,Z 411.417,A -85,B 0,C 180,E1 16238.308,E2 16238.308} C_VEL
LIN {X 0,Y 290.368,Z 406.705,A -85,B 0,C 180,E1 16239.07,E2 16239.07} C_VEL
LIN {X 0,Y 291.932,Z 407.26,A -85,B 0,C 180,E1 16239.518,E2 16239.518} C_VEL
LIN {X 0,Y 303.878,Z 432.849,A -85,B 0,C 180,E1 16244.399,E2 16244.399} C_VEL
LIN {X 0,Y 311.677,Z 458.575,A -85,B 0,C 180,E1 16248.75,E2 16248.75} C_VEL
LIN {X 0,Y 313.078,Z 468.148,A -85,B 0,C 180,E1 16250.254,E2 16250.254} C_VEL
LIN {X 0,Y 304.127,Z 498.631,A -85,B 0,C 180,E1 16253.768,E2 16253.768} C_VEL
LIN {X 0,Y 294.56,Z 524.899,A -85,B 0,C 180,E1 16258.303,E2 16258.303} C_VEL
LIN {X 0,Y 285.314,Z 547.364,A -85,B 0,C 180,E1 16264.044,E2 16264.044} C_VEL
LIN {X 0,Y 278.502,Z 563.228,A -85,B 0,C 180,E1 16270.143,E2 16270.143} C_VEL
LIN {X 0,Y 273.965,Z 574.884,A -85,B 0,C 180,E1 16277.235,E2 16277.235} C_VEL
LIN {X 0,Y 272.06,Z 580.591,A -85,B 0,C 180,E1 16283.615,E2 16283.615} C_VEL
LIN {X 0,Y 271.418,Z 582.434,A -85,B 0,C 180,E1 16290.005,E2 16290.005} C_VEL
LIN {X 0,Y 272.376,Z 579.417,A -85,B 0,C 180,E1 16297.992,E2 16297.992} C_VEL
LIN {X 0,Y 275.24,Z 571.466,A -85,B 0,C 180,E1 16305.15,E2 16305.15} C_VEL
LIN {X 0,Y 280.901,Z 557.662,A -85,B 0,C 180,E1 16312.17,E2 16312.17} C_VEL
LIN {X 0,Y 288.652,Z 539.34,A -85,B 0,C 180,E1 16318.172,E2 16318.172} C_VEL
LIN {X 0,Y 297.911,Z 515.953,A -85,B 0,C 180,E1 16323.33,E2 16323.33} C_VEL
LIN {X 0,Y 307.581,Z 487.651,A -85,B 0,C 180,E1 16327.54,E2 16327.54} C_VEL
LIN {X 0,Y 313.112,Z 466.484,A -85,B 0,C 180,E1 16329.844,E2 16329.844} C_VEL
LIN {X 0,Y 306.393,Z 440.044,A -85,B 0,C 180,E1 16334.238,E2 16334.238} C_VEL
LIN {X 0,Y 294.61,Z 412.197,A -85,B 0,C 180,E1 16339.312,E2 16339.312} C_VEL
LIN {X 0,Y 280.305,Z 389.204,A -85,B 0,C 180,E1 16344.669,E2 16344.669} C_VEL
LIN {X 0,Y 271.729,Z 376.823,A -85,B 0,C 180,E1 16348.219,E2 16348.219} C_VEL
LIN {X 0,Y 268.406,Z 372.194,A -85,B 0,C 180,E1 16349.763,E2 16349.763} C_VEL
LIN {X 0,Y 268.119,Z 370.16,A -85,B 0,C 180,E1 16349.993,E2 16349.993} C_VEL
LIN {X 0,Y 268.365,Z 370.16,A -85,B 0,C 180,E1 16356.744,E2 16356.744} C_VEL
LIN {X 0,Y 268.923,Z 370.16,A -85,B 0,C 180,E1 16363.654,E2 16363.654} C_VEL
LIN {X 0,Y 269.391,Z 370.16,A -85,B 0,C 180,E1 16371.498,E2 16371.498} C_VEL
LIN {X 0,Y 270.281,Z 370.16,A -85,B 0,C 180,E1 16380.002,E2 16380.002} C_VEL
LIN {X 0,Y 269.626,Z 370.16,A -85,B 0,C 180,E1 16386.45,E2 16386.45} C_VEL
LIN {X 0,Y 269.074,Z 370.16,A -85,B 0,C 180,E1 16393.008,E2 16393.008} C_VEL
LIN {X 0,Y 268.62,Z 370.16,A -85,B 0,C 180,E1 16399.767,E2 16399.767} C_VEL
LIN {X 0,Y 268.228,Z 370.175,A -85,B 0,C 180,E1 16404.907,E2 16404.907} C_VEL
LIN {X 0,Y 270.13,Z 375.225,A -85,B 0,C 180,E1 16405.962,E2 16405.962} C_VEL
LIN {X 0,Y 273.283,Z 378.758,A -85,B 0,C 180,E1 16407.344,E2 16407.344} C_VEL
LIN {X 0,Y 287.025,Z 399.38,A -85,B 0,C 180,E1 16412.74,E2 16412.74} C_VEL
LIN {X 0,Y 300.334,Z 422.503,A -85,B 0,C 180,E1 16417.337,E2 16417.337} C_VEL
LIN {X 0,Y 311.344,Z 449.682,A -85,B 0,C 180,E1 16421.636,E2 16421.636} C_VEL
LIN {X 0,Y 315.555,Z 466.681,A -85,B 0,C 180,E1 16423.969,E2 16423.969} C_VEL
LIN {X 0,Y 306.857,Z 502.445,A -85,B 0,C 180,E1 16426.953,E2 16426.953} C_VEL
LIN {X 0,Y 297.287,Z 534.112,A -85,B 0,C 180,E1 16430.93,E2 16430.93} C_VEL
LIN {X 0,Y 287.826,Z 562.092,A -85,B 0,C 180,E1 16436.017,E2 16436.017} C_VEL
LIN {X 0,Y 279.711,Z 585.688,A -85,B 0,C 180,E1 16442.166,E2 16442.166} C_VEL
LIN {X 0,Y 274.263,Z 603.659,A -85,B 0,C 180,E1 16448.876,E2 16448.876} C_VEL
LIN {X 0,Y 271.518,Z 616.835,A -85,B 0,C 180,E1 16456.287,E2 16456.287} C_VEL
LIN {X 0,Y 270.94,Z 624.184,A -85,B 0,C 180,E1 16463.579,E2 16463.579} C_VEL
LIN {X 0,Y 271.068,Z 626.326,A -85,B 0,C 180,E1 16469.995,E2 16469.995} C_VEL
LIN {X 0,Y 270.935,Z 624.201,A -85,B 0,C 180,E1 16476.412,E2 16476.412} C_VEL
LIN {X 0,Y 271.539,Z 616.871,A -85,B 0,C 180,E1 16483.702,E2 16483.702} C_VEL
LIN {X 0,Y 274.251,Z 603.731,A -85,B 0,C 180,E1 16491.118,E2 16491.118} C_VEL
LIN {X 0,Y 280.044,Z 584.521,A -85,B 0,C 180,E1 16498.226,E2 16498.226} C_VEL
LIN {X 0,Y 292.129,Z 552.394,A -85,B 0,C 180,E1 16506.31,E2 16506.31} C_VEL
LIN {X 0,Y 307.76,Z 518.255,A -85,B 0,C 180,E1 16512.343,E2 16512.343} C_VEL
LIN {X 0,Y 323.785,Z 486.56,A -85,B 0,C 180,E1 16516.174,E2 16516.174} C_VEL
LIN {X 0,Y 331.516,Z 471.293,A -85,B 0,C 180,E1 16517.645,E2 16517.645} C_VEL
LIN {X 0,Y 332.252,Z 470.133,A -85,B 0,C 180,E1 16518.094,E2 16518.094} C_VEL
LIN {X 0,Y 318.048,Z 501.334,A -85,B 0,C 180,E1 16521.552,E2 16521.552} C_VEL
LIN {X 0,Y 311.37,Z 515.045,A -85,B 0,C 180,E1 16523.578,E2 16523.578} C_VEL
LIN {X 0,Y 302.984,Z 528.138,A -85,B 0,C 180,E1 16525.135,E2 16525.135} C_VEL
LIN {X 0,Y 295.29,Z 538.767,A -85,B 0,C 180,E1 16526.625,E2 16526.625} C_VEL
LIN {X 0,Y 294.48,Z 540.079,A -85,B 0,C 180,E1 16526.919,E2 16526.919} C_VEL
LIN {X 0,Y 282.779,Z 559.621,A -85,B 0,C 180,E1 16532.641,E2 16532.641} C_VEL
LIN {X 0,Y 273.884,Z 573.588,A -85,B 0,C 180,E1 16538.941,E2 16538.941} C_VEL
LIN {X 0,Y 268.269,Z 581.817,A -85,B 0,C 180,E1 16545.287,E2 16545.287} C_VEL
LIN {X 0,Y 265.687,Z 584.866,A -85,B 0,C 180,E1 16550.155,E2 16550.155} C_VEL
LIN {X 0,Y 264.039,Z 584.878,A -85,B 0,C 180,E1 16556.711,E2 16556.711} C_VEL
LIN {X 0,Y 263.453,Z 580.185,A -85,B 0,C 180,E1 16563.292,E2 16563.292} C_VEL
LIN {X 0,Y 264.249,Z 570.256,A -85,B 0,C 180,E1 16569.895,E2 16569.895} C_VEL
LIN {X 0,Y 266.323,Z 554.264,A -85,B 0,C 180,E1 16576.51,E2 16576.51} C_VEL
LIN {X 0,Y 269.967,Z 533.183,A -85,B 0,C 180,E1 16582.434,E2 16582.434} C_VEL
LIN {X 0,Y 274.785,Z 506.533,A -85,B 0,C 180,E1 16587.699,E2 16587.699} C_VEL
LIN {X 0,Y 280.121,Z 475.097,A -85,B 0,C 180,E1 16592.024,E2 16592.024} C_VEL
LIN {X 0,Y 283.907,Z 444.014,A -85,B 0,C 180,E1 16595.015,E2 16595.015} C_VEL
LIN {X 0,Y 278.703,Z 423.724,A -85,B 0,C 180,E1 16597.165,E2 16597.165} C_VEL
LIN {X 0,Y 282.417,Z 422.445,A -85,B 0,C 180,E1 16598.124,E2 16598.124} C_VEL
LIN {X 0,Y 286.466,Z 418.891,A -85,B 0,C 180,E1 16598.928,E2 16598.928} C_VEL
LIN {X 0,Y 289.583,Z 416.508,A -85,B 0,C 180,E1 16599.577,E2 16599.577} C_VEL
LIN {X 0,Y 300.292,Z 442.358,A -85,B 0,C 180,E1 16604.6,E2 16604.6} C_VEL
LIN {X 0,Y 306.465,Z 466.78,A -85,B 0,C 180,E1 16608.877,E2 16608.877} C_VEL
LIN {X 0,Y 305.948,Z 473.364,A -85,B 0,C 180,E1 16609.737,E2 16609.737} C_VEL
LIN {X 0,Y 296.62,Z 502.769,A -85,B 0,C 180,E1 16613.384,E2 16613.384} C_VEL
LIN {X 0,Y 286.678,Z 528.628,A -85,B 0,C 180,E1 16618.129,E2 16618.129} C_VEL
LIN {X 0,Y 277.197,Z 550.328,A -85,B 0,C 180,E1 16624.097,E2 16624.097} C_VEL
LIN {X 0,Y 269.769,Z 566.976,A -85,B 0,C 180,E1 16631.18,E2 16631.18} C_VEL
LIN {X 0,Y 265.561,Z 577.324,A -85,B 0,C 180,E1 16638.495,E2 16638.495} C_VEL
LIN {X 0,Y 264.231,Z 581.228,A -85,B 0,C 180,E1 16643.425,E2 16643.425} C_VEL
LIN {X 0,Y 263.543,Z 583.071,A -85,B 0,C 180,E1 16650.005,E2 16650.005} C_VEL
LIN {X 0,Y 264.575,Z 580.055,A -85,B 0,C 180,E1 16658.229,E2 16658.229} C_VEL
LIN {X 0,Y 267.9,Z 571.288,A -85,B 0,C 180,E1 16666.13,E2 16666.13} C_VEL
LIN {X 0,Y 273.576,Z 558.32,A -85,B 0,C 180,E1 16672.796,E2 16672.796} C_VEL
LIN {X 0,Y 282.285,Z 538.619,A -85,B 0,C 180,E1 16679.305,E2 16679.305} C_VEL
LIN {X 0,Y 291.987,Z 515.185,A -85,B 0,C 180,E1 16684.456,E2 16684.456} C_VEL
LIN {X 0,Y 301.837,Z 487.021,A -85,B 0,C 180,E1 16688.626,E2 16688.626} C_VEL
LIN {X 0,Y 306.763,Z 469.496,A -85,B 0,C 180,E1 16690.543,E2 16690.543} C_VEL
LIN {X 0,Y 300.953,Z 444.724,A -85,B 0,C 180,E1 16694.859,E2 16694.859} C_VEL
LIN {X 0,Y 290.163,Z 417.663,A -85,B 0,C 180,E1 16700.032,E2 16700.032} C_VEL
LIN {X 0,Y 276.916,Z 395.362,A -85,B 0,C 180,E1 16705.446,E2 16705.446} C_VEL
LIN {X 0,Y 268.442,Z 383.211,A -85,B 0,C 180,E1 16709.154,E2 16709.154} C_VEL
LIN {X 0,Y 264.281,Z 377.044,A -85,B 0,C 180,E1 16711.239,E2 16711.239} C_VEL
LIN {X 0,Y 260.618,Z 372.338,A -85,B 0,C 180,E1 16713.222,E2 16713.222} C_VEL
LIN {X 0,Y 260.309,Z 370.16,A -85,B 0,C 180,E1 16713.732,E2 16713.732} C_VEL
LIN {X 0,Y 260.941,Z 370.16,A -85,B 0,C 180,E1 16723.139,E2 16723.139} C_VEL
LIN {X 0,Y 261.451,Z 370.16,A -85,B 0,C 180,E1 16731.524,E2 16731.524} C_VEL
LIN {X 0,Y 262.373,Z 370.16,A -85,B 0,C 180,E1 16740.002,E2 16740.002} C_VEL
LIN {X 0,Y 261.679,Z 370.16,A -85,B 0,C 180,E1 16746.647,E2 16746.647} C_VEL
LIN {X 0,Y 261.107,Z 370.16,A -85,B 0,C 180,E1 16753.412,E2 16753.412} C_VEL
LIN {X 0,Y 260.5,Z 370.75,A -85,B 0,C 180,E1 16761.482,E2 16761.482} C_VEL
LIN {X 0,Y 262.798,Z 375.768,A -85,B 0,C 180,E1 16762.903,E2 16762.903} C_VEL
LIN {X 0,Y 265.728,Z 378.986,A -85,B 0,C 180,E1 16764.392,E2 16764.392} C_VEL
LIN {X 0,Y 275.968,Z 393.904,A -85,B 0,C 180,E1 16769.077,E2 16769.077} C_VEL
LIN {X 0,Y 290.06,Z 416.54,A -85,B 0,C 180,E1 16774.472,E2 16774.472} C_VEL
LIN {X 0,Y 301.911,Z 442.512,A -85,B 0,C 180,E1 16779.164,E2 16779.164} C_VEL
LIN {X 0,Y 309.481,Z 468.194,A -85,B 0,C 180,E1 16783.069,E2 16783.069} C_VEL
LIN {X 0,Y 300.378,Z 503.67,A -85,B 0,C 180,E1 16786.125,E2 16786.125} C_VEL
LIN {X 0,Y 290.247,Z 535.682,A -85,B 0,C 180,E1 16790.28,E2 16790.28} C_VEL
LIN {X 0,Y 280.47,Z 563.038,A -85,B 0,C 180,E1 16795.469,E2 16795.469} C_VEL
LIN {X 0,Y 272.093,Z 586.261,A -85,B 0,C 180,E1 16801.769,E2 16801.769} C_VEL
LIN {X 0,Y 266.275,Z 604.466,A -85,B 0,C 180,E1 16808.949,E2 16808.949} C_VEL
LIN {X 0,Y 263.579,Z 617.234,A -85,B 0,C 180,E1 16816.713,E2 16816.713} C_VEL
LIN {X 0,Y 263.047,Z 623.54,A -85,B 0,C 180,E1 16823.385,E2 16823.385} C_VEL
LIN {X 0,Y 263.188,Z 625.689,A -85,B 0,C 180,E1 16829.995,E2 16829.995} C_VEL
LIN {X 0,Y 263.042,Z 623.558,A -85,B 0,C 180,E1 16836.605,E2 16836.605} C_VEL
LIN {X 0,Y 263.747,Z 616.233,A -85,B 0,C 180,E1 16844.115,E2 16844.115} C_VEL
LIN {X 0,Y 267.199,Z 601.624,A -85,B 0,C 180,E1 16852.48,E2 16852.48} C_VEL
LIN {X 0,Y 274.815,Z 580.538,A -85,B 0,C 180,E1 16860.405,E2 16860.405} C_VEL
LIN {X 0,Y 287.864,Z 551.463,A -85,B 0,C 180,E1 16867.964,E2 16867.964} C_VEL
LIN {X 0,Y 305.435,Z 518.265,A -85,B 0,C 180,E1 16873.936,E2 16873.936} C_VEL
LIN {X 0,Y 323.737,Z 486.509,A -85,B 0,C 180,E1 16877.754,E2 16877.754} C_VEL
LIN {X 0,Y 324.374,Z 485.525,A -85,B 0,C 180,E1 16878.083,E2 16878.083} C_VEL
LIN {X 0,Y 307.264,Z 517.685,A -85,B 0,C 180,E1 16882.424,E2 16882.424} C_VEL
LIN {X 0,Y 294.48,Z 540.079,A -85,B 0,C 180,E1 16886.919,E2 16886.919} C_VEL
LIN {X 0,Y 285.749,Z 551.118,A -85,B 0,C 180,E1 16889.015,E2 16889.015} C_VEL
LIN {X 0,Y 277.943,Z 559.791,A -85,B 0,C 180,E1 16891.018,E2 16891.018} C_VEL
LIN {X 0,Y 277.186,Z 560.815,A -85,B 0,C 180,E1 16891.38,E2 16891.38} C_VEL
LIN {X 0,Y 266.748,Z 575.479,A -85,B 0,C 180,E1 16898.35,E2 16898.35} C_VEL
LIN {X 0,Y 260.737,Z 583.195,A -85,B 0,C 180,E1 16904.852,E2 16904.852} C_VEL
LIN {X 0,Y 257.961,Z 585.88,A -85,B 0,C 180,E1 16909.857,E2 16909.857} C_VEL
LIN {X 0,Y 256.186,Z 585.538,A -85,B 0,C 180,E1 16916.61,E2 16916.61} C_VEL
LIN {X 0,Y 255.577,Z 580.413,A -85,B 0,C 180,E1 16923.394,E2 16923.394} C_VEL
LIN {X 0,Y 256.409,Z 570.133,A -85,B 0,C 180,E1 16930.2,E2 16930.2} C_VEL
LIN {X 0,Y 258.638,Z 553.65,A -85,B 0,C 180,E1 16937.016,E2 16937.016} C_VEL
LIN {X 0,Y 262.354,Z 532.682,A -85,B 0,C 180,E1 16942.948,E2 16942.948} C_VEL
LIN {X 0,Y 267.41,Z 505.373,A -85,B 0,C 180,E1 16948.374,E2 16948.374} C_VEL
LIN {X 0,Y 272.886,Z 473.691,A -85,B 0,C 180,E1 16952.743,E2 16952.743} C_VEL
LIN {X 0,Y 276.237,Z 444.781,A -85,B 0,C 180,E1 16955.584,E2 16955.584} C_VEL
LIN {X 0,Y 273.587,Z 434.045,A -85,B 0,C 180,E1 16956.749,E2 16956.749} C_VEL
LIN {X 0,Y 275.06,Z 434.473,A -85,B 0,C 180,E1 16957.257,E2 16957.257} C_VEL
LIN {X 0,Y 287.05,Z 426.042,A -85,B 0,C 180,E1 16959.75,E2 16959.75} C_VEL
LIN {X 0,Y 296.339,Z 451.942,A -85,B 0,C 180,E1 16964.878,E2 16964.878} C_VEL
LIN {X 0,Y 300.44,Z 472.573,A -85,B 0,C 180,E1 16968.602,E2 16968.602} C_VEL
LIN {X 0,Y 290.752,Z 502.394,A -85,B 0,C 180,E1 16972.285,E2 16972.285} C_VEL
LIN {X 0,Y 280.665,Z 527.682,A -85,B 0,C 180,E1 16976.911,E2 16976.911} C_VEL
LIN {X 0,Y 271.169,Z 548.688,A -85,B 0,C 180,E1 16982.58,E2 16982.58} C_VEL
LIN {X 0,Y 263.644,Z 564.529,A -85,B 0,C 180,E1 16988.973,E2 16988.973} C_VEL
LIN {X 0,Y 258.572,Z 576.163,A -85,B 0,C 180,E1 16996.461,E2 16996.461} C_VEL
LIN {X 0,Y 256.393,Z 581.865,A -85,B 0,C 180,E1 17003.223,E2 17003.223} C_VEL
LIN {X 0,Y 255.691,Z 583.706,A -85,B 0,C 180,E1 17010.005,E2 17010.005} C_VEL
LIN {X 0,Y 256.776,Z 580.695,A -85,B 0,C 180,E1 17018.481,E2 17018.481} C_VEL
LIN {X 0,Y 260.023,Z 572.616,A -85,B 0,C 180,E1 17026.162,E2 17026.162} C_VEL
LIN {X 0,Y 266.291,Z 558.975,A -85,B 0,C 180,E1 17033.456,E2 17033.456} C_VEL
LIN {X 0,Y 275.407,Z 539.303,A -85,B 0,C 180,E1 17040.112,E2 17040.112} C_VEL
LIN {X 0,Y 285.638,Z 515.626,A -85,B 0,C 180,E1 17045.403,E2 17045.403} C_VEL
LIN {X 0,Y 295.758,Z 487.746,A -85,B 0,C 180,E1 17049.588,E2 17049.588} C_VEL
LIN {X 0,Y 300.401,Z 471.909,A -85,B 0,C 180,E1 17051.371,E2 17051.371} C_VEL
LIN {X 0,Y 294.687,Z 446.732,A -85,B 0,C 180,E1 17055.998,E2 17055.998} C_VEL
LIN {X 0,Y 284.511,Z 420.664,A -85,B 0,C 180,E1 17061.304,E2 17061.304} C_VEL
LIN {X 0,Y 271.04,Z 397.226,A -85,B 0,C 180,E1 17067.382,E2 17067.382} C_VEL
LIN {X 0,Y 261.332,Z 383.735,A -85,B 0,C 180,E1 17072.168,E2 17072.168} C_VEL
LIN {X 0,Y 256.611,Z 377.112,A -85,B 0,C 180,E1 17074.955,E2 17074.955} C_VEL
LIN {X 0,Y 252.813,Z 372.401,A -85,B 0,C 180,E1 17077.513,E2 17077.513} C_VEL
LIN {X 0,Y 252.533,Z 370.16,A -85,B 0,C 180,E1 17078.023,E2 17078.023} C_VEL
LIN {X 0,Y 253.21,Z 370.16,A -85,B 0,C 180,E1 17086.166,E2 17086.166} C_VEL
LIN {X 0,Y 253.791,Z 370.16,A -85,B 0,C 180,E1 17093.15,E2 17093.15} C_VEL
LIN {X 0,Y 254.47,Z 370.16,A -85,B 0,C 180,E1 17100.002,E2 17100.002} C_VEL
LIN {X 0,Y 253.758,Z 370.16,A -85,B 0,C 180,E1 17106.855,E2 17106.855} C_VEL
LIN {X 0,Y 253.12,Z 370.16,A -85,B 0,C 180,E1 17113.844,E2 17113.844} C_VEL
LIN {X 0,Y 252.914,Z 370.96,A -85,B 0,C 180,E1 17117.305,E2 17117.305} C_VEL
LIN {X 0,Y 255.181,Z 375.906,A -85,B 0,C 180,E1 17119.047,E2 17119.047} C_VEL
LIN {X 0,Y 258.146,Z 378.759,A -85,B 0,C 180,E1 17120.857,E2 17120.857} C_VEL
LIN {X 0,Y 262.372,Z 384.399,A -85,B 0,C 180,E1 17123.262,E2 17123.262} C_VEL
LIN {X 0,Y 275.815,Z 404.784,A -85,B 0,C 180,E1 17129.606,E2 17129.606} C_VEL
LIN {X 0,Y 288.878,Z 428.125,A -85,B 0,C 180,E1 17134.976,E2 17134.976} C_VEL
LIN {X 0,Y 299.159,Z 454.456,A -85,B 0,C 180,E1 17139.686,E2 17139.686} C_VEL
LIN {X 0,Y 303.03,Z 471.537,A -85,B 0,C 180,E1 17142.285,E2 17142.285} C_VEL
LIN {X 0,Y 293.685,Z 505.933,A -85,B 0,C 180,E1 17145.377,E2 17145.377} C_VEL
LIN {X 0,Y 283.188,Z 537.181,A -85,B 0,C 180,E1 17149.607,E2 17149.607} C_VEL
LIN {X 0,Y 273.148,Z 563.984,A -85,B 0,C 180,E1 17154.892,E2 17154.892} C_VEL
LIN {X 0,Y 264.471,Z 586.832,A -85,B 0,C 180,E1 17161.347,E2 17161.347} C_VEL
LIN {X 0,Y 258.58,Z 604.233,A -85,B 0,C 180,E1 17168.53,E2 17168.53} C_VEL
LIN {X 0,Y 255.735,Z 616.576,A -85,B 0,C 180,E1 17176.297,E2 17176.297} C_VEL
LIN {X 0,Y 255.154,Z 622.896,A -85,B 0,C 180,E1 17183.18,E2 17183.18} C_VEL
LIN {X 0,Y 255.323,Z 625.053,A -85,B 0,C 180,E1 17189.995,E2 17189.995} C_VEL
LIN {X 0,Y 255.149,Z 622.915,A -85,B 0,C 180,E1 17196.81,E2 17196.81} C_VEL
LIN {X 0,Y 255.94,Z 615.748,A -85,B 0,C 180,E1 17204.555,E2 17204.555} C_VEL
LIN {X 0,Y 259.176,Z 603.627,A -85,B 0,C 180,E1 17212.309,E2 17212.309} C_VEL
LIN {X 0,Y 267.186,Z 583.577,A -85,B 0,C 180,E1 17220.655,E2 17220.655} C_VEL
LIN {X 0,Y 281.756,Z 554.833,A -85,B 0,C 180,E1 17228.762,E2 17228.762} C_VEL
LIN {X 0,Y 300.659,Z 523.324,A -85,B 0,C 180,E1 17234.82,E2 17234.82} C_VEL
LIN {X 0,Y 315.852,Z 500,A -85,B 0,C 180,E1 17237.93,E2 17237.93} C_VEL
LIN {X 0,Y 313.631,Z 503.793,A -85,B 0,C 180,E1 17238.688,E2 17238.688} C_VEL
LIN {X 0,Y 295.97,Z 532.38,A -85,B 0,C 180,E1 17243.512,E2 17243.512} C_VEL
LIN {X 0,Y 281.368,Z 554.674,A -85,B 0,C 180,E1 17249.259,E2 17249.259} C_VEL
LIN {X 0,Y 277.186,Z 560.815,A -85,B 0,C 180,E1 17251.38,E2 17251.38} C_VEL
LIN {X 0,Y 268.748,Z 569.305,A -85,B 0,C 180,E1 17254.085,E2 17254.085} C_VEL
LIN {X 0,Y 260.546,Z 576.363,A -85,B 0,C 180,E1 17257.056,E2 17257.056} C_VEL
LIN {X 0,Y 253.2,Z 584.518,A -85,B 0,C 180,E1 17264.389,E2 17264.389} C_VEL
LIN {X 0,Y 250.236,Z 586.91,A -85,B 0,C 180,E1 17269.541,E2 17269.541} C_VEL
LIN {X 0,Y 248.316,Z 586.132,A -85,B 0,C 180,E1 17276.502,E2 17276.502} C_VEL
LIN {X 0,Y 247.686,Z 580.604,A -85,B 0,C 180,E1 17283.502,E2 17283.502} C_VEL
LIN {X 0,Y 248.573,Z 569.921,A -85,B 0,C 180,E1 17290.525,E2 17290.525} C_VEL
LIN {X 0,Y 250.741,Z 554.179,A -85,B 0,C 180,E1 17297.116,E2 17297.116} C_VEL
LIN {X 0,Y 254.67,Z 532.529,A -85,B 0,C 180,E1 17303.367,E2 17303.367} C_VEL
LIN {X 0,Y 259.803,Z 505.653,A -85,B 0,C 180,E1 17308.826,E2 17308.826} C_VEL
LIN {X 0,Y 265.456,Z 474.033,A -85,B 0,C 180,E1 17313.29,E2 17313.29} C_VEL
LIN {X 0,Y 269.075,Z 447.58,A -85,B 0,C 180,E1 17315.946,E2 17315.946} C_VEL
LIN {X 0,Y 268.427,Z 444.085,A -85,B 0,C 180,E1 17316.461,E2 17316.461} C_VEL
LIN {X 0,Y 276.948,Z 440.235,A -85,B 0,C 180,E1 17318.52,E2 17318.52} C_VEL
LIN {X 0,Y 283.555,Z 435.767,A -85,B 0,C 180,E1 17319.84,E2 17319.84} C_VEL
LIN {X 0,Y 289.617,Z 452.19,A -85,B 0,C 180,E1 17323.395,E2 17323.395} C_VEL
LIN {X 0,Y 294.112,Z 475.257,A -85,B 0,C 180,E1 17327.779,E2 17327.779} C_VEL
LIN {X 0,Y 284.14,Z 504.262,A -85,B 0,C 180,E1 17331.491,E2 17331.491} C_VEL
LIN {X 0,Y 273.373,Z 530.005,A -85,B 0,C 180,E1 17336.378,E2 17336.378} C_VEL
LIN {X 0,Y 263.054,Z 551.654,A -85,B 0,C 180,E1 17342.592,E2 17342.592} C_VEL
LIN {X 0,Y 254.787,Z 568.273,A -85,B 0,C 180,E1 17350.027,E2 17350.027} C_VEL
LIN {X 0,Y 250.105,Z 578.605,A -85,B 0,C 180,E1 17357.774,E2 17357.774} C_VEL
LIN {X 0,Y 248.572,Z 582.502,A -85,B 0,C 180,E1 17363.009,E2 17363.009} C_VEL
LIN {X 0,Y 247.815,Z 584.343,A -85,B 0,C 180,E1 17370.005,E2 17370.005} C_VEL
LIN {X 0,Y 248.979,Z 581.333,A -85,B 0,C 180,E1 17378.749,E2 17378.749} C_VEL
LIN {X 0,Y 252.093,Z 574.044,A -85,B 0,C 180,E1 17386.092,E2 17386.092} C_VEL
LIN {X 0,Y 258.138,Z 561.486,A -85,B 0,C 180,E1 17393.326,E2 17393.326} C_VEL
LIN {X 0,Y 267.326,Z 542.741,A -85,B 0,C 180,E1 17400.179,E2 17400.179} C_VEL
LIN {X 0,Y 277.478,Z 520.434,A -85,B 0,C 180,E1 17405.549,E2 17405.549} C_VEL
LIN {X 0,Y 287.972,Z 493.676,A -85,B 0,C 180,E1 17409.924,E2 17409.924} C_VEL
LIN {X 0,Y 294.045,Z 474.037,A -85,B 0,C 180,E1 17412.291,E2 17412.291} C_VEL
LIN {X 0,Y 288.741,Z 449.486,A -85,B 0,C 180,E1 17417.033,E2 17417.033} C_VEL
LIN {X 0,Y 279.261,Z 424.56,A -85,B 0,C 180,E1 17422.422,E2 17422.422} C_VEL
LIN {X 0,Y 267.288,Z 402.932,A -85,B 0,C 180,E1 17428.407,E2 17428.407} C_VEL
LIN {X 0,Y 258.641,Z 390.385,A -85,B 0,C 180,E1 17433.029,E2 17433.029} C_VEL
LIN {X 0,Y 254.296,Z 384.269,A -85,B 0,C 180,E1 17435.725,E2 17435.725} C_VEL
LIN {X 0,Y 250.48,Z 378.555,A -85,B 0,C 180,E1 17438.508,E2 17438.508} C_VEL
LIN {X 0,Y 245.597,Z 372.917,A -85,B 0,C 180,E1 17442.797,E2 17442.797} C_VEL
LIN {X 0,Y 245.135,Z 370.16,A -85,B 0,C 180,E1 17443.585,E2 17443.585} C_VEL
LIN {X 0,Y 245.837,Z 370.16,A -85,B 0,C 180,E1 17452.928,E2 17452.928} C_VEL
LIN {X 0,Y 246.56,Z 370.16,A -85,B 0,C 180,E1 17460.002,E2 17460.002} C_VEL
LIN {X 0,Y 245.55,Z 370.16,A -85,B 0,C 180,E1 17469.403,E2 17469.403} C_VEL
LIN {X 0,Y 245.341,Z 370.467,A -85,B 0,C 180,E1 17471.571,E2 17471.571} C_VEL
LIN {X 0,Y 247.001,Z 375.136,A -85,B 0,C 180,E1 17473.516,E2 17473.516} C_VEL
LIN {X 0,Y 250.848,Z 378.808,A -85,B 0,C 180,E1 17476.658,E2 17476.658} C_VEL
LIN {X 0,Y 254.523,Z 384.296,A -85,B 0,C 180,E1 17479.323,E2 17479.323} C_VEL
LIN {X 0,Y 264.943,Z 398.95,A -85,B 0,C 180,E1 17485.265,E2 17485.265} C_VEL
LIN {X 0,Y 278.269,Z 421.013,A -85,B 0,C 180,E1 17491.465,E2 17491.465} C_VEL
LIN {X 0,Y 289.718,Z 446.651,A -85,B 0,C 180,E1 17496.808,E2 17496.808} C_VEL
LIN {X 0,Y 296.943,Z 472.314,A -85,B 0,C 180,E1 17501.218,E2 17501.218} C_VEL
LIN {X 0,Y 287.509,Z 506.622,A -85,B 0,C 180,E1 17504.419,E2 17504.419} C_VEL
LIN {X 0,Y 276.975,Z 536.607,A -85,B 0,C 180,E1 17508.551,E2 17508.551} C_VEL
LIN {X 0,Y 266.54,Z 563.263,A -85,B 0,C 180,E1 17513.887,E2 17513.887} C_VEL
LIN {X 0,Y 257.345,Z 586.137,A -85,B 0,C 180,E1 17520.477,E2 17520.477} C_VEL
LIN {X 0,Y 251.015,Z 603.561,A -85,B 0,C 180,E1 17527.849,E2 17527.849} C_VEL
LIN {X 0,Y 247.917,Z 615.919,A -85,B 0,C 180,E1 17535.856,E2 17535.856} C_VEL
LIN {X 0,Y 247.263,Z 622.252,A -85,B 0,C 180,E1 17542.961,E2 17542.961} C_VEL
LIN {X 0,Y 247.442,Z 624.415,A -85,B 0,C 180,E1 17549.995,E2 17549.995} C_VEL
LIN {X 0,Y 247.258,Z 622.272,A -85,B 0,C 180,E1 17557.029,E2 17557.029} C_VEL
LIN {X 0,Y 248.377,Z 614.497,A -85,B 0,C 180,E1 17565.914,E2 17565.914} C_VEL
LIN {X 0,Y 253.112,Z 600.617,A -85,B 0,C 180,E1 17574.746,E2 17574.746} C_VEL
LIN {X 0,Y 262.492,Z 581.036,A -85,B 0,C 180,E1 17582.867,E2 17582.867} C_VEL
LIN {X 0,Y 278.649,Z 553.65,A -85,B 0,C 180,E1 17590.684,E2 17590.684} C_VEL
LIN {X 0,Y 298.642,Z 524.638,A -85,B 0,C 180,E1 17596.351,E2 17596.351} C_VEL
LIN {X 0,Y 306.983,Z 513.182,A -85,B 0,C 180,E1 17598.025,E2 17598.025} C_VEL
LIN {X 0,Y 305.907,Z 514.9,A -85,B 0,C 180,E1 17598.586,E2 17598.586} C_VEL
LIN {X 0,Y 287.521,Z 541.003,A -85,B 0,C 180,E1 17603.673,E2 17603.673} C_VEL
LIN {X 0,Y 272.057,Z 561.832,A -85,B 0,C 180,E1 17609.943,E2 17609.943} C_VEL
LIN {X 0,Y 260.546,Z 576.363,A -85,B 0,C 180,E1 17617.056,E2 17617.056} C_VEL
LIN {X 0,Y 252.692,Z 581.974,A -85,B 0,C 180,E1 17620.336,E2 17620.336} C_VEL
LIN {X 0,Y 246.154,Z 585.566,A -85,B 0,C 180,E1 17623.412,E2 17623.412} C_VEL
LIN {X 0,Y 245.696,Z 585.869,A -85,B 0,C 180,E1 17623.905,E2 17623.905} C_VEL
LIN {X 0,Y 242.539,Z 587.923,A -85,B 0,C 180,E1 17629.205,E2 17629.205} C_VEL
LIN {X 0,Y 240.449,Z 586.669,A -85,B 0,C 180,E1 17636.388,E2 17636.388} C_VEL
LIN {X 0,Y 239.796,Z 580.793,A -85,B 0,C 180,E1 17643.617,E2 17643.617} C_VEL
LIN {X 0,Y 240.744,Z 569.573,A -85,B 0,C 180,E1 17650.872,E2 17650.872} C_VEL
LIN {X 0,Y 243.08,Z 553.435,A -85,B 0,C 180,E1 17657.672,E2 17657.672} C_VEL
LIN {X 0,Y 247.347,Z 530.629,A -85,B 0,C 180,E1 17664.237,E2 17664.237} C_VEL
LIN {X 0,Y 252.614,Z 503.772,A -85,B 0,C 180,E1 17669.654,E2 17669.654} C_VEL
LIN {X 0,Y 258.319,Z 472.326,A -85,B 0,C 180,E1 17674.082,E2 17674.082} C_VEL
LIN {X 0,Y 261.087,Z 455.753,A -85,B 0,C 180,E1 17675.923,E2 17675.923} C_VEL
LIN {X 0,Y 265.49,Z 453.776,A -85,B 0,C 180,E1 17677.037,E2 17677.037} C_VEL
LIN {X 0,Y 268.314,Z 451.013,A -85,B 0,C 180,E1 17677.467,E2 17677.467} C_VEL
LIN {X 0,Y 280.848,Z 445.43,A -85,B 0,C 180,E1 17680.302,E2 17680.302} C_VEL
LIN {X 0,Y 286.988,Z 470.414,A -85,B 0,C 180,E1 17685.498,E2 17685.498} C_VEL
LIN {X 0,Y 287.521,Z 478.489,A -85,B 0,C 180,E1 17686.985,E2 17686.985} C_VEL
LIN {X 0,Y 277.146,Z 507.253,A -85,B 0,C 180,E1 17690.837,E2 17690.837} C_VEL
LIN {X 0,Y 266.073,Z 532.236,A -85,B 0,C 180,E1 17695.82,E2 17695.82} C_VEL
LIN {X 0,Y 256.044,Z 552.316,A -85,B 0,C 180,E1 17701.775,E2 17701.775} C_VEL
LIN {X 0,Y 247.343,Z 568.919,A -85,B 0,C 180,E1 17709.399,E2 17709.399} C_VEL
LIN {X 0,Y 242.404,Z 579.245,A -85,B 0,C 180,E1 17717.379,E2 17717.379} C_VEL
LIN {X 0,Y 240.746,Z 583.139,A -85,B 0,C 180,E1 17722.78,E2 17722.78} C_VEL
LIN {X 0,Y 239.941,Z 584.981,A -85,B 0,C 180,E1 17730.005,E2 17730.005} C_VEL
LIN {X 0,Y 241.179,Z 581.972,A -85,B 0,C 180,E1 17739.034,E2 17739.034} C_VEL
LIN {X 0,Y 244.508,Z 574.686,A -85,B 0,C 180,E1 17746.606,E2 17746.606} C_VEL
LIN {X 0,Y 250.904,Z 562.141,A -85,B 0,C 180,E1 17754.04,E2 17754.04} C_VEL
LIN {X 0,Y 260.522,Z 543.41,A -85,B 0,C 180,E1 17761.053,E2 17761.053} C_VEL
LIN {X 0,Y 271.726,Z 519.724,A -85,B 0,C 180,E1 17766.8,E2 17766.8} C_VEL
LIN {X 0,Y 282.999,Z 491.807,A -85,B 0,C 180,E1 17771.299,E2 17771.299} C_VEL
LIN {X 0,Y 287.765,Z 476.626,A -85,B 0,C 180,E1 17773.158,E2 17773.158} C_VEL
LIN {X 0,Y 282.708,Z 451.926,A -85,B 0,C 180,E1 17778.178,E2 17778.178} C_VEL
LIN {X 0,Y 274.114,Z 428.475,A -85,B 0,C 180,E1 17783.582,E2 17783.582} C_VEL
LIN {X 0,Y 263.345,Z 408.251,A -85,B 0,C 180,E1 17789.526,E2 17789.526} C_VEL
LIN {X 0,Y 255.741,Z 396.694,A -85,B 0,C 180,E1 17794.014,E2 17794.014} C_VEL
LIN {X 0,Y 252.02,Z 391.298,A -85,B 0,C 180,E1 17796.515,E2 17796.515} C_VEL
LIN {X 0,Y 247.634,Z 384.858,A -85,B 0,C 180,E1 17799.933,E2 17799.933} C_VEL
LIN {X 0,Y 243.927,Z 380.055,A -85,B 0,C 180,E1 17803.512,E2 17803.512} C_VEL
LIN {X 0,Y 243.019,Z 377.767,A -85,B 0,C 180,E1 17804.696,E2 17804.696} C_VEL
LIN {X 0,Y 238.09,Z 371.35,A -85,B 0,C 180,E1 17814.644,E2 17814.644} C_VEL
LIN {X 0,Y 238.265,Z 370.16,A -85,B 0,C 180,E1 17816.359,E2 17816.359} C_VEL
LIN {X 0,Y 238.447,Z 370.979,A -85,B 0,C 180,E1 17821.48,E2 17821.48} C_VEL
LIN {X 0,Y 241.722,Z 377.048,A -85,B 0,C 180,E1 17828.668,E2 17828.668} C_VEL
LIN {X 0,Y 243.66,Z 378.579,A -85,B 0,C 180,E1 17830.971,E2 17830.971} C_VEL
LIN {X 0,Y 246.963,Z 384.21,A -85,B 0,C 180,E1 17834.423,E2 17834.423} C_VEL
LIN {X 0,Y 249.009,Z 386.412,A -85,B 0,C 180,E1 17836.107,E2 17836.107} C_VEL
LIN {X 0,Y 254.833,Z 395.234,A -85,B 0,C 180,E1 17840.316,E2 17840.316} C_VEL
LIN {X 0,Y 262.8,Z 406.847,A -85,B 0,C 180,E1 17844.916,E2 17844.916} C_VEL
LIN {X 0,Y 274.795,Z 427.913,A -85,B 0,C 180,E1 17850.984,E2 17850.984} C_VEL
LIN {X 0,Y 285.076,Z 452.801,A -85,B 0,C 180,E1 17856.345,E2 17856.345} C_VEL
LIN {X 0,Y 290.825,Z 475.019,A -85,B 0,C 180,E1 17860.322,E2 17860.322} C_VEL
LIN {X 0,Y 280.424,Z 510.136,A -85,B 0,C 180,E1 17863.767,E2 17863.767} C_VEL
LIN {X 0,Y 268.894,Z 540.991,A -85,B 0,C 180,E1 17868.306,E2 17868.306} C_VEL
LIN {X 0,Y 257.384,Z 568.649,A -85,B 0,C 180,E1 17874.386,E2 17874.386} C_VEL
LIN {X 0,Y 248.004,Z 590.99,A -85,B 0,C 180,E1 17881.655,E2 17881.655} C_VEL
LIN {X 0,Y 242.059,Z 607.471,A -85,B 0,C 180,E1 17889.749,E2 17889.749} C_VEL
LIN {X 0,Y 239.729,Z 617.683,A -85,B 0,C 180,E1 17897.663,E2 17897.663} C_VEL
LIN {X 0,Y 239.387,Z 621.609,A -85,B 0,C 180,E1 17902.728,E2 17902.728} C_VEL
LIN {X 0,Y 239.569,Z 623.778,A -85,B 0,C 180,E1 17909.995,E2 17909.995} C_VEL
LIN {X 0,Y 239.383,Z 621.63,A -85,B 0,C 180,E1 17917.261,E2 17917.261} C_VEL
LIN {X 0,Y 240.645,Z 614.296,A -85,B 0,C 180,E1 17926.44,E2 17926.44} C_VEL
LIN {X 0,Y 245.819,Z 601.114,A -85,B 0,C 180,E1 17935.532,E2 17935.532} C_VEL
LIN {X 0,Y 256.169,Z 582.295,A -85,B 0,C 180,E1 17943.921,E2 17943.921} C_VEL
LIN {X 0,Y 273.194,Z 556.826,A -85,B 0,C 180,E1 17951.675,E2 17951.675} C_VEL
LIN {X 0,Y 295.073,Z 528.576,A -85,B 0,C 180,E1 17957.496,E2 17957.496} C_VEL
LIN {X 0,Y 297.798,Z 525.253,A -85,B 0,C 180,E1 17958.047,E2 17958.047} C_VEL
LIN {X 0,Y 298.288,Z 524.676,A -85,B 0,C 180,E1 17958.423,E2 17958.423} C_VEL
LIN {X 0,Y 277.973,Z 550.165,A -85,B 0,C 180,E1 17964.161,E2 17964.161} C_VEL
LIN {X 0,Y 262.707,Z 568.261,A -85,B 0,C 180,E1 17970.668,E2 17970.668} C_VEL
LIN {X 0,Y 251.521,Z 580.389,A -85,B 0,C 180,E1 17977.9,E2 17977.9} C_VEL
LIN {X 0,Y 245.696,Z 585.869,A -85,B 0,C 180,E1 17983.905,E2 17983.905} C_VEL
LIN {X 0,Y 243.111,Z 587.12,A -85,B 0,C 180,E1 17985.849,E2 17985.849} C_VEL
LIN {X 0,Y 233.948,Z 588.796,A -85,B 0,C 180,E1 17991.228,E2 17991.228} C_VEL
LIN {X 0,Y 233.695,Z 588.67,A -85,B 0,C 180,E1 17991.763,E2 17991.763} C_VEL
LIN {X 0,Y 232.144,Z 584.64,A -85,B 0,C 180,E1 17999.998,E2 17999.998} C_VEL
LIN {X 0,Y 232.28,Z 575.785,A -85,B 0,C 180,E1 18007.487,E2 18007.487} C_VEL
LIN {X 0,Y 234.071,Z 561.066,A -85,B 0,C 180,E1 18014.991,E2 18014.991} C_VEL
LIN {X 0,Y 237.685,Z 540.677,A -85,B 0,C 180,E1 18021.972,E2 18021.972} C_VEL
LIN {X 0,Y 242.828,Z 514.848,A -85,B 0,C 180,E1 18028.128,E2 18028.128} C_VEL
LIN {X 0,Y 248.805,Z 484.06,A -85,B 0,C 180,E1 18033.201,E2 18033.201} C_VEL
LIN {X 0,Y 251.787,Z 468.789,A -85,B 0,C 180,E1 18035.234,E2 18035.234} C_VEL
LIN {X 0,Y 257.35,Z 466.03,A -85,B 0,C 180,E1 18036.621,E2 18036.621} C_VEL
LIN {X 0,Y 262.508,Z 462.001,A -85,B 0,C 180,E1 18037.529,E2 18037.529} C_VEL
LIN {X 0,Y 267.807,Z 457.894,A -85,B 0,C 180,E1 18038.447,E2 18038.447} C_VEL
LIN {X 0,Y 276.748,Z 453.975,A -85,B 0,C 180,E1 18040.4,E2 18040.4} C_VEL
LIN {X 0,Y 281.385,Z 476.87,A -85,B 0,C 180,E1 18045.334,E2 18045.334} C_VEL
LIN {X 0,Y 281.107,Z 481.498,A -85,B 0,C 180,E1 18046.14,E2 18046.14} C_VEL
LIN {X 0,Y 269.731,Z 511.166,A -85,B 0,C 180,E1 18050.33,E2 18050.33} C_VEL
LIN {X 0,Y 257.758,Z 536.608,A -85,B 0,C 180,E1 18055.777,E2 18055.777} C_VEL
LIN {X 0,Y 247.204,Z 556.43,A -85,B 0,C 180,E1 18062.258,E2 18062.258} C_VEL
LIN {X 0,Y 239.202,Z 571.015,A -85,B 0,C 180,E1 18069.635,E2 18069.635} C_VEL
LIN {X 0,Y 234.685,Z 579.887,A -85,B 0,C 180,E1 18076.957,E2 18076.957} C_VEL
LIN {X 0,Y 232.93,Z 583.776,A -85,B 0,C 180,E1 18082.537,E2 18082.537} C_VEL
LIN {X 0,Y 232.066,Z 585.618,A -85,B 0,C 180,E1 18090.006,E2 18090.006} C_VEL
LIN {X 0,Y 233.392,Z 582.611,A -85,B 0,C 180,E1 18099.338,E2 18099.338} C_VEL
LIN {X 0,Y 237.357,Z 574.536,A -85,B 0,C 180,E1 18107.769,E2 18107.769} C_VEL
LIN {X 0,Y 244.691,Z 560.939,A -85,B 0,C 180,E1 18115.67,E2 18115.67} C_VEL
LIN {X 0,Y 255.169,Z 541.346,A -85,B 0,C 180,E1 18122.784,E2 18122.784} C_VEL
LIN {X 0,Y 266.352,Z 518.573,A -85,B 0,C 180,E1 18128.185,E2 18128.185} C_VEL
LIN {X 0,Y 277.502,Z 491.569,A -85,B 0,C 180,E1 18132.507,E2 18132.507} C_VEL
LIN {X 0,Y 281.491,Z 479.005,A -85,B 0,C 180,E1 18134.096,E2 18134.096} C_VEL
LIN {X 0,Y 277.167,Z 455.857,A -85,B 0,C 180,E1 18139.049,E2 18139.049} C_VEL
LIN {X 0,Y 269.648,Z 433.842,A -85,B 0,C 180,E1 18144.377,E2 18144.377} C_VEL
LIN {X 0,Y 259.635,Z 413.755,A -85,B 0,C 180,E1 18150.564,E2 18150.564} C_VEL
LIN {X 0,Y 250.658,Z 399.16,A -85,B 0,C 180,E1 18156.63,E2 18156.63} C_VEL
LIN {X 0,Y 245.444,Z 391.982,A -85,B 0,C 180,E1 18160.911,E2 18160.911} C_VEL
LIN {X 0,Y 242.021,Z 386.196,A -85,B 0,C 180,E1 18164.631,E2 18164.631} C_VEL
LIN {X 0,Y 237.084,Z 378.122,A -85,B 0,C 180,E1 18175.768,E2 18175.768} C_VEL
LIN {X 0,Y 237.363,Z 378.675,A -85,B 0,C 180,E1 18181.03,E2 18181.03} C_VEL
LIN {X 0,Y 240.66,Z 384.877,A -85,B 0,C 180,E1 18188.595,E2 18188.595} C_VEL
LIN {X 0,Y 242.235,Z 386.594,A -85,B 0,C 180,E1 18190.581,E2 18190.581} C_VEL
LIN {X 0,Y 246.244,Z 392.357,A -85,B 0,C 180,E1 18194.693,E2 18194.693} C_VEL
LIN {X 0,Y 255.632,Z 406.407,A -85,B 0,C 180,E1 18201.612,E2 18201.612} C_VEL
LIN {X 0,Y 266.491,Z 425.356,A -85,B 0,C 180,E1 18207.951,E2 18207.951} C_VEL
LIN {X 0,Y 276.066,Z 446.5,A -85,B 0,C 180,E1 18213.259,E2 18213.259} C_VEL
LIN {X 0,Y 283.347,Z 470.742,A -85,B 0,C 180,E1 18218.135,E2 18218.135} C_VEL
LIN {X 0,Y 284.623,Z 478.869,A -85,B 0,C 180,E1 18219.532,E2 18219.532} C_VEL
LIN {X 0,Y 273.898,Z 512.152,A -85,B 0,C 180,E1 18222.907,E2 18222.907} C_VEL
LIN {X 0,Y 261.999,Z 542.37,A -85,B 0,C 180,E1 18227.512,E2 18227.512} C_VEL
LIN {X 0,Y 250.308,Z 568.961,A -85,B 0,C 180,E1 18233.579,E2 18233.579} C_VEL
LIN {X 0,Y 240.944,Z 589.929,A -85,B 0,C 180,E1 18240.581,E2 18240.581} C_VEL
LIN {X 0,Y 234.446,Z 606.805,A -85,B 0,C 180,E1 18249.061,E2 18249.061} C_VEL
LIN {X 0,Y 231.966,Z 616.625,A -85,B 0,C 180,E1 18256.792,E2 18256.792} C_VEL
LIN {X 0,Y 231.498,Z 620.965,A -85,B 0,C 180,E1 18262.479,E2 18262.479} C_VEL
LIN {X 0,Y 231.687,Z 623.14,A -85,B 0,C 180,E1 18269.994,E2 18269.994} C_VEL
LIN {X 0,Y 231.494,Z 620.986,A -85,B 0,C 180,E1 18277.51,E2 18277.51} C_VEL
LIN {X 0,Y 232.919,Z 614.139,A -85,B 0,C 180,E1 18287.001,E2 18287.001} C_VEL
LIN {X 0,Y 238.6,Z 601.663,A -85,B 0,C 180,E1 18296.363,E2 18296.363} C_VEL
LIN {X 0,Y 250.792,Z 582.349,A -85,B 0,C 180,E1 18305.483,E2 18305.483} C_VEL
LIN {X 0,Y 269.965,Z 557.399,A -85,B 0,C 180,E1 18313.384,E2 18313.384} C_VEL
LIN {X 0,Y 288.955,Z 535.613,A -85,B 0,C 180,E1 18318.153,E2 18318.153} C_VEL
LIN {X 0,Y 288.387,Z 536.313,A -85,B 0,C 180,E1 18318.754,E2 18318.754} C_VEL
LIN {X 0,Y 268.362,Z 558.334,A -85,B 0,C 180,E1 18324.671,E2 18324.671} C_VEL
LIN {X 0,Y 253.368,Z 573.916,A -85,B 0,C 180,E1 18331.442,E2 18331.442} C_VEL
LIN {X 0,Y 243.372,Z 583.153,A -85,B 0,C 180,E1 18338.082,E2 18338.082} C_VEL
LIN {X 0,Y 236.979,Z 588.024,A -85,B 0,C 180,E1 18345.192,E2 18345.192} C_VEL
LIN {X 0,Y 233.695,Z 588.67,A -85,B 0,C 180,E1 18351.763,E2 18351.763} C_VEL
LIN {X 0,Y 230.454,Z 588.065,A -85,B 0,C 180,E1 18354.898,E2 18354.898} C_VEL
LIN {X 0,Y 224.391,Z 585.221,A -85,B 0,C 180,E1 18359.626,E2 18359.626} C_VEL
LIN {X 0,Y 224.215,Z 584.719,A -85,B 0,C 180,E1 18360.174,E2 18360.174} C_VEL
LIN {X 0,Y 224.439,Z 575.571,A -85,B 0,C 180,E1 18367.751,E2 18367.751} C_VEL
LIN {X 0,Y 226.329,Z 560.397,A -85,B 0,C 180,E1 18375.516,E2 18375.516} C_VEL
LIN {X 0,Y 230.126,Z 539.823,A -85,B 0,C 180,E1 18382.575,E2 18382.575} C_VEL
LIN {X 0,Y 235.462,Z 513.749,A -85,B 0,C 180,E1 18388.827,E2 18388.827} C_VEL
LIN {X 0,Y 241.658,Z 482.378,A -85,B 0,C 180,E1 18394.046,E2 18394.046} C_VEL
LIN {X 0,Y 242.294,Z 480.402,A -85,B 0,C 180,E1 18394.486,E2 18394.486} C_VEL
LIN {X 0,Y 246.498,Z 478.893,A -85,B 0,C 180,E1 18395.691,E2 18395.691} C_VEL
LIN {X 0,Y 258.361,Z 470.962,A -85,B 0,C 180,E1 18397.968,E2 18397.968} C_VEL
LIN {X 0,Y 270.372,Z 462.973,A -85,B 0,C 180,E1 18400.082,E2 18400.082} C_VEL
LIN {X 0,Y 272.559,Z 463.23,A -85,B 0,C 180,E1 18400.738,E2 18400.738} C_VEL
LIN {X 0,Y 275.271,Z 482.995,A -85,B 0,C 180,E1 18405.084,E2 18405.084} C_VEL
LIN {X 0,Y 263.718,Z 511.889,A -85,B 0,C 180,E1 18409.238,E2 18409.238} C_VEL
LIN {X 0,Y 251.597,Z 536.675,A -85,B 0,C 180,E1 18414.607,E2 18414.607} C_VEL
LIN {X 0,Y 241.077,Z 555.673,A -85,B 0,C 180,E1 18420.794,E2 18420.794} C_VEL
LIN {X 0,Y 231.777,Z 571.663,A -85,B 0,C 180,E1 18428.952,E2 18428.952} C_VEL
LIN {X 0,Y 227.001,Z 580.527,A -85,B 0,C 180,E1 18436.507,E2 18436.507} C_VEL
LIN {X 0,Y 225.1,Z 584.415,A -85,B 0,C 180,E1 18442.275,E2 18442.275} C_VEL
LIN {X 0,Y 224.218,Z 586.253,A -85,B 0,C 180,E1 18450.006,E2 18450.006} C_VEL
LIN {X 0,Y 225.616,Z 583.249,A -85,B 0,C 180,E1 18459.663,E2 18459.663} C_VEL
LIN {X 0,Y 229.466,Z 575.871,A -85,B 0,C 180,E1 18467.821,E2 18467.821} C_VEL
LIN {X 0,Y 236.521,Z 563.453,A -85,B 0,C 180,E1 18475.604,E2 18475.604} C_VEL
LIN {X 0,Y 247.118,Z 544.75,A -85,B 0,C 180,E1 18482.943,E2 18482.943} C_VEL
LIN {X 0,Y 259.296,Z 521.152,A -85,B 0,C 180,E1 18488.883,E2 18488.883} C_VEL
LIN {X 0,Y 271.204,Z 493.879,A -85,B 0,C 180,E1 18493.427,E2 18493.427} C_VEL
LIN {X 0,Y 275.264,Z 481.228,A -85,B 0,C 180,E1 18495.114,E2 18495.114} C_VEL
LIN {X 0,Y 271.42,Z 458.854,A -85,B 0,C 180,E1 18500.176,E2 18500.176} C_VEL
LIN {X 0,Y 265.155,Z 439.161,A -85,B 0,C 180,E1 18505.186,E2 18505.186} C_VEL
LIN {X 0,Y 255.608,Z 418.472,A -85,B 0,C 180,E1 18511.829,E2 18511.829} C_VEL
LIN {X 0,Y 247.567,Z 405.447,A -85,B 0,C 180,E1 18517.888,E2 18517.888} C_VEL
LIN {X 0,Y 243.689,Z 399.42,A -85,B 0,C 180,E1 18521.452,E2 18521.452} C_VEL
LIN {X 0,Y 240.046,Z 393.067,A -85,B 0,C 180,E1 18525.849,E2 18525.849} C_VEL
LIN {X 0,Y 236.071,Z 385.788,A -85,B 0,C 180,E1 18536.326,E2 18536.326} C_VEL
LIN {X 0,Y 236.318,Z 386.605,A -85,B 0,C 180,E1 18540.805,E2 18540.805} C_VEL
LIN {X 0,Y 239.682,Z 392.752,A -85,B 0,C 180,E1 18548.63,E2 18548.63} C_VEL
LIN {X 0,Y 240.997,Z 394.892,A -85,B 0,C 180,E1 18550.407,E2 18550.407} C_VEL
LIN {X 0,Y 245.7,Z 402.062,A -85,B 0,C 180,E1 18555.298,E2 18555.298} C_VEL
LIN {X 0,Y 253.153,Z 413.526,A -85,B 0,C 180,E1 18561.03,E2 18561.03} C_VEL
LIN {X 0,Y 263.22,Z 432.278,A -85,B 0,C 180,E1 18567.467,E2 18567.467} C_VEL
LIN {X 0,Y 271.76,Z 452.898,A -85,B 0,C 180,E1 18572.796,E2 18572.796} C_VEL
LIN {X 0,Y 278.129,Z 476.948,A -85,B 0,C 180,E1 18577.779,E2 18577.779} C_VEL
LIN {X 0,Y 278.382,Z 481.848,A -85,B 0,C 180,E1 18578.593,E2 18578.593} C_VEL
LIN {X 0,Y 266.895,Z 515.568,A -85,B 0,C 180,E1 18582.18,E2 18582.18} C_VEL
LIN {X 0,Y 254.686,Z 544.606,A -85,B 0,C 180,E1 18586.868,E2 18586.868} C_VEL
LIN {X 0,Y 242.728,Z 570.57,A -85,B 0,C 180,E1 18593.1,E2 18593.1} C_VEL
LIN {X 0,Y 232.684,Z 591.956,A -85,B 0,C 180,E1 18600.771,E2 18600.771} C_VEL
LIN {X 0,Y 226.287,Z 607.872,A -85,B 0,C 180,E1 18609.5,E2 18609.5} C_VEL
LIN {X 0,Y 223.888,Z 617.694,A -85,B 0,C 180,E1 18618.29,E2 18618.29} C_VEL
LIN {X 0,Y 223.58,Z 621.897,A -85,B 0,C 180,E1 18626.112,E2 18626.112} C_VEL
LIN {X 0,Y 223.818,Z 622.503,A -85,B 0,C 180,E1 18629.994,E2 18629.994} C_VEL
LIN {X 0,Y 223.63,Z 620.344,A -85,B 0,C 180,E1 18637.776,E2 18637.776} C_VEL
LIN {X 0,Y 225.187,Z 613.973,A -85,B 0,C 180,E1 18647.604,E2 18647.604} C_VEL
LIN {X 0,Y 231.436,Z 602.174,A -85,B 0,C 180,E1 18657.246,E2 18657.246} C_VEL
LIN {X 0,Y 244.853,Z 583.65,A -85,B 0,C 180,E1 18666.696,E2 18666.696} C_VEL
LIN {X 0,Y 265.93,Z 559.527,A -85,B 0,C 180,E1 18674.783,E2 18674.783} C_VEL
LIN {X 0,Y 278.703,Z 546.279,A -85,B 0,C 180,E1 18677.982,E2 18677.982} C_VEL
LIN {X 0,Y 280.272,Z 544.693,A -85,B 0,C 180,E1 18678.641,E2 18678.641} C_VEL
LIN {X 0,Y 259.528,Z 564.828,A -85,B 0,C 180,E1 18684.889,E2 18684.889} C_VEL
LIN {X 0,Y 243.85,Z 578.918,A -85,B 0,C 180,E1 18692.247,E2 18692.247} C_VEL
LIN {X 0,Y 234.218,Z 586.389,A -85,B 0,C 180,E1 18699.173,E2 18699.173} C_VEL
LIN {X 0,Y 229.413,Z 589.25,A -85,B 0,C 180,E1 18704.692,E2 18704.692} C_VEL
LIN {X 0,Y 225.692,Z 589.284,A -85,B 0,C 180,E1 18712.288,E2 18712.288} C_VEL
LIN {X 0,Y 224.215,Z 584.719,A -85,B 0,C 180,E1 18720.174,E2 18720.174} C_VEL
LIN {X 0,Y 222.762,Z 582.679,A -85,B 0,C 180,E1 18722.317,E2 18722.317} C_VEL
LIN {X 0,Y 216.668,Z 575.109,A -85,B 0,C 180,E1 18728.14,E2 18728.14} C_VEL
LIN {X 0,Y 216.669,Z 574.251,A -85,B 0,C 180,E1 18728.681,E2 18728.681} C_VEL
LIN {X 0,Y 218.821,Z 558.251,A -85,B 0,C 180,E1 18736.579,E2 18736.579} C_VEL
LIN {X 0,Y 223.114,Z 536.053,A -85,B 0,C 180,E1 18744.021,E2 18744.021} C_VEL
LIN {X 0,Y 228.864,Z 509.083,A -85,B 0,C 180,E1 18750.259,E2 18750.259} C_VEL
LIN {X 0,Y 232.782,Z 490.416,A -85,B 0,C 180,E1 18753.556,E2 18753.556} C_VEL
LIN {X 0,Y 239.07,Z 487.937,A -85,B 0,C 180,E1 18755.351,E2 18755.351} C_VEL
LIN {X 0,Y 257.445,Z 477.359,A -85,B 0,C 180,E1 18759.052,E2 18759.052} C_VEL
LIN {X 0,Y 267.455,Z 470.433,A -85,B 0,C 180,E1 18760.61,E2 18760.61} C_VEL
LIN {X 0,Y 269.046,Z 485.914,A -85,B 0,C 180,E1 18764.156,E2 18764.156} C_VEL
LIN {X 0,Y 256.811,Z 514.664,A -85,B 0,C 180,E1 18768.462,E2 18768.462} C_VEL
LIN {X 0,Y 244.352,Z 538.906,A -85,B 0,C 180,E1 18773.964,E2 18773.964} C_VEL
LIN {X 0,Y 232.792,Z 558.591,A -85,B 0,C 180,E1 18780.813,E2 18780.813} C_VEL
LIN {X 0,Y 223.6,Z 573.655,A -85,B 0,C 180,E1 18789.184,E2 18789.184} C_VEL
LIN {X 0,Y 218.457,Z 582.685,A -85,B 0,C 180,E1 18798.007,E2 18798.007} C_VEL
LIN {X 0,Y 216.442,Z 586.407,A -85,B 0,C 180,E1 18805.995,E2 18805.995} C_VEL
LIN {X 0,Y 216.46,Z 586.37,A -85,B 0,C 180,E1 18814.017,E2 18814.017} C_VEL
LIN {X 0,Y 218.522,Z 582.572,A -85,B 0,C 180,E1 18822.002,E2 18822.002} C_VEL
LIN {X 0,Y 223.691,Z 573.471,A -85,B 0,C 180,E1 18830.819,E2 18830.819} C_VEL
LIN {X 0,Y 232.703,Z 558.682,A -85,B 0,C 180,E1 18839.009,E2 18839.009} C_VEL
LIN {X 0,Y 244.65,Z 538.151,A -85,B 0,C 180,E1 18846.132,E2 18846.132} C_VEL
LIN {X 0,Y 257.46,Z 513.057,A -85,B 0,C 180,E1 18851.705,E2 18851.705} C_VEL
LIN {X 0,Y 269.216,Z 484.556,A -85,B 0,C 180,E1 18855.933,E2 18855.933} C_VEL
LIN {X 0,Y 265.548,Z 461.138,A -85,B 0,C 180,E1 18861.51,E2 18861.51} C_VEL
LIN {X 0,Y 259.61,Z 441.867,A -85,B 0,C 180,E1 18866.804,E2 18866.804} C_VEL
LIN {X 0,Y 251.481,Z 423.626,A -85,B 0,C 180,E1 18873.169,E2 18873.169} C_VEL
LIN {X 0,Y 245.063,Z 412.346,A -85,B 0,C 180,E1 18878.636,E2 18878.636} C_VEL
LIN {X 0,Y 241.419,Z 406.428,A -85,B 0,C 180,E1 18882.384,E2 18882.384} C_VEL
LIN {X 0,Y 238.292,Z 400.6,A -85,B 0,C 180,E1 18886.662,E2 18886.662} C_VEL
LIN {X 0,Y 235.069,Z 393.837,A -85,B 0,C 180,E1 18896.31,E2 18896.31} C_VEL
LIN {X 0,Y 235.295,Z 394.592,A -85,B 0,C 180,E1 18900.694,E2 18900.694} C_VEL
LIN {X 0,Y 239.31,Z 401.974,A -85,B 0,C 180,E1 18909.676,E2 18909.676} C_VEL
LIN {X 0,Y 244.079,Z 410.035,A -85,B 0,C 180,E1 18915.057,E2 18915.057} C_VEL
LIN {X 0,Y 250.93,Z 421.392,A -85,B 0,C 180,E1 18920.762,E2 18920.762} C_VEL
LIN {X 0,Y 259.692,Z 439.021,A -85,B 0,C 180,E1 18926.979,E2 18926.979} C_VEL
LIN {X 0,Y 267.917,Z 461.201,A -85,B 0,C 180,E1 18932.806,E2 18932.806} C_VEL
LIN {X 0,Y 272.685,Z 482.76,A -85,B 0,C 180,E1 18937.393,E2 18937.393} C_VEL
LIN {X 0,Y 261.004,Z 516.067,A -85,B 0,C 180,E1 18941.05,E2 18941.05} C_VEL
LIN {X 0,Y 247.88,Z 545.848,A -85,B 0,C 180,E1 18945.987,E2 18945.987} C_VEL
LIN {X 0,Y 235.507,Z 571.371,A -85,B 0,C 180,E1 18952.353,E2 18952.353} C_VEL
LIN {X 0,Y 225.081,Z 592.344,A -85,B 0,C 180,E1 18960.256,E2 18960.256} C_VEL
LIN {X 0,Y 218.237,Z 608.539,A -85,B 0,C 180,E1 18969.699,E2 18969.699} C_VEL
LIN {X 0,Y 215.899,Z 617.898,A -85,B 0,C 180,E1 18979.034,E2 18979.034} C_VEL
LIN {X 0,Y 215.681,Z 621.256,A -85,B 0,C 180,E1 18985.969,E2 18985.969} C_VEL
LIN {X 0,Y 215.934,Z 621.866,A -85,B 0,C 180,E1 18989.994,E2 18989.994} C_VEL
LIN {X 0,Y 215.742,Z 619.7,A -85,B 0,C 180,E1 18998.062,E2 18998.062} C_VEL
LIN {X 0,Y 217.495,Z 613.748,A -85,B 0,C 180,E1 19008.248,E2 19008.248} C_VEL
LIN {X 0,Y 224.351,Z 602.772,A -85,B 0,C 180,E1 19018.181,E2 19018.181} C_VEL
LIN {X 0,Y 239.32,Z 584.661,A -85,B 0,C 180,E1 19028.112,E2 19028.112} C_VEL
LIN {X 0,Y 261.577,Z 562.183,A -85,B 0,C 180,E1 19036.094,E2 19036.094} C_VEL
LIN {X 0,Y 270.9,Z 553.514,A -85,B 0,C 180,E1 19038.365,E2 19038.365} C_VEL
LIN {X 0,Y 267.788,Z 556.237,A -85,B 0,C 180,E1 19039.603,E2 19039.603} C_VEL
LIN {X 0,Y 247.134,Z 573.568,A -85,B 0,C 180,E1 19046.539,E2 19046.539} C_VEL
LIN {X 0,Y 231.627,Z 585.114,A -85,B 0,C 180,E1 19054.857,E2 19054.857} C_VEL
LIN {X 0,Y 224.884,Z 589.127,A -85,B 0,C 180,E1 19060.456,E2 19060.456} C_VEL
LIN {X 0,Y 219.437,Z 590.732,A -85,B 0,C 180,E1 19068.052,E2 19068.052} C_VEL
LIN {X 0,Y 216.844,Z 588.091,A -85,B 0,C 180,E1 19075.994,E2 19075.994} C_VEL
LIN {X 0,Y 216.127,Z 580.844,A -85,B 0,C 180,E1 19084.014,E2 19084.014} C_VEL
LIN {X 0,Y 216.669,Z 574.251,A -85,B 0,C 180,E1 19088.681,E2 19088.681} C_VEL
LIN {X 0,Y 214.811,Z 568.793,A -85,B 0,C 180,E1 19091.812,E2 19091.812} C_VEL
LIN {X 0,Y 210.895,Z 559.228,A -85,B 0,C 180,E1 19096.392,E2 19096.392} C_VEL
LIN {X 0,Y 210.997,Z 558.019,A -85,B 0,C 180,E1 19096.898,E2 19096.898} C_VEL
LIN {X 0,Y 215.423,Z 535.641,A -85,B 0,C 180,E1 19104.512,E2 19104.512} C_VEL
LIN {X 0,Y 221.637,Z 507.471,A -85,B 0,C 180,E1 19111.126,E2 19111.126} C_VEL
LIN {X 0,Y 223.294,Z 499.799,A -85,B 0,C 180,E1 19112.641,E2 19112.641} C_VEL
LIN {X 0,Y 228.243,Z 498.353,A -85,B 0,C 180,E1 19114.316,E2 19114.316} C_VEL
LIN {X 0,Y 233.685,Z 495.707,A -85,B 0,C 180,E1 19115.663,E2 19115.663} C_VEL
LIN {X 0,Y 255.492,Z 484.204,A -85,B 0,C 180,E1 19120.039,E2 19120.039} C_VEL
LIN {X 0,Y 261.467,Z 480.021,A -85,B 0,C 180,E1 19120.859,E2 19120.859} C_VEL
LIN {X 0,Y 262.961,Z 483.111,A -85,B 0,C 180,E1 19121.962,E2 19121.962} C_VEL
LIN {X 0,Y 262.478,Z 489.634,A -85,B 0,C 180,E1 19123.309,E2 19123.309} C_VEL
LIN {X 0,Y 249.995,Z 517.434,A -85,B 0,C 180,E1 19127.653,E2 19127.653} C_VEL
LIN {X 0,Y 236.708,Z 541.719,A -85,B 0,C 180,E1 19133.475,E2 19133.475} C_VEL
LIN {X 0,Y 224.679,Z 561.301,A -85,B 0,C 180,E1 19140.763,E2 19140.763} C_VEL
LIN {X 0,Y 215.419,Z 575.561,A -85,B 0,C 180,E1 19149.434,E2 19149.434} C_VEL
LIN {X 0,Y 210.754,Z 583.322,A -85,B 0,C 180,E1 19157.561,E2 19157.561} C_VEL
LIN {X 0,Y 208.582,Z 587.044,A -85,B 0,C 180,E1 19165.844,E2 19165.844} C_VEL
LIN {X 0,Y 208.601,Z 587.008,A -85,B 0,C 180,E1 19174.168,E2 19174.168} C_VEL
LIN {X 0,Y 210.814,Z 583.212,A -85,B 0,C 180,E1 19182.448,E2 19182.448} C_VEL
LIN {X 0,Y 216.29,Z 574.117,A -85,B 0,C 180,E1 19191.566,E2 19191.566} C_VEL
LIN {X 0,Y 226.061,Z 558.943,A -85,B 0,C 180,E1 19200.157,E2 19200.157} C_VEL
LIN {X 0,Y 238.076,Z 539.243,A -85,B 0,C 180,E1 19207.133,E2 19207.133} C_VEL
LIN {X 0,Y 251.12,Z 514.815,A -85,B 0,C 180,E1 19212.713,E2 19212.713} C_VEL
LIN {X 0,Y 263.137,Z 487.654,A -85,B 0,C 180,E1 19216.823,E2 19216.823} C_VEL
LIN {X 0,Y 260.219,Z 465.676,A -85,B 0,C 180,E1 19222.326,E2 19222.326} C_VEL
LIN {X 0,Y 255.014,Z 447.004,A -85,B 0,C 180,E1 19227.707,E2 19227.707} C_VEL
LIN {X 0,Y 247.524,Z 428.825,A -85,B 0,C 180,E1 19234.411,E2 19234.411} C_VEL
LIN {X 0,Y 241.953,Z 418.433,A -85,B 0,C 180,E1 19239.828,E2 19239.828} C_VEL
LIN {X 0,Y 239.202,Z 413.49,A -85,B 0,C 180,E1 19243.137,E2 19243.137} C_VEL
LIN {X 0,Y 236.705,Z 408.253,A -85,B 0,C 180,E1 19247.033,E2 19247.033} C_VEL
LIN {X 0,Y 233.939,Z 401.894,A -85,B 0,C 180,E1 19256.292,E2 19256.292} C_VEL
LIN {X 0,Y 234.175,Z 402.897,A -85,B 0,C 180,E1 19260.928,E2 19260.928} C_VEL
LIN {X 0,Y 237.723,Z 409.653,A -85,B 0,C 180,E1 19269.279,E2 19269.279} C_VEL
LIN {X 0,Y 241.963,Z 417.477,A -85,B 0,C 180,E1 19274.612,E2 19274.612} C_VEL
LIN {X 0,Y 248.225,Z 428.769,A -85,B 0,C 180,E1 19280.358,E2 19280.358} C_VEL
LIN {X 0,Y 255.813,Z 445.255,A -85,B 0,C 180,E1 19286.323,E2 19286.323} C_VEL
LIN {X 0,Y 263.039,Z 466.647,A -85,B 0,C 180,E1 19292.158,E2 19292.158} C_VEL
LIN {X 0,Y 266.727,Z 485.403,A -85,B 0,C 180,E1 19296.332,E2 19296.332} C_VEL
LIN {X 0,Y 254.32,Z 518.614,A -85,B 0,C 180,E1 19300.152,E2 19300.152} C_VEL
LIN {X 0,Y 241.135,Z 547.091,A -85,B 0,C 180,E1 19305.057,E2 19305.057} C_VEL
LIN {X 0,Y 228.322,Z 572.069,A -85,B 0,C 180,E1 19311.558,E2 19311.558} C_VEL
LIN {X 0,Y 217.501,Z 592.694,A -85,B 0,C 180,E1 19319.686,E2 19319.686} C_VEL
LIN {X 0,Y 210.495,Z 608.239,A -85,B 0,C 180,E1 19329.232,E2 19329.232} C_VEL
LIN {X 0,Y 208.002,Z 617.53,A -85,B 0,C 180,E1 19339.055,E2 19339.055} C_VEL
LIN {X 0,Y 207.79,Z 620.616,A -85,B 0,C 180,E1 19345.816,E2 19345.816} C_VEL
LIN {X 0,Y 208.049,Z 621.228,A -85,B 0,C 180,E1 19349.994,E2 19349.994} C_VEL
LIN {X 0,Y 207.848,Z 619.055,A -85,B 0,C 180,E1 19358.37,E2 19358.37} C_VEL
LIN {X 0,Y 210.802,Z 611.926,A -85,B 0,C 180,E1 19371.038,E2 19371.038} C_VEL
LIN {X 0,Y 221.05,Z 598.858,A -85,B 0,C 180,E1 19382.344,E2 19382.344} C_VEL
LIN {X 0,Y 243.056,Z 577.275,A -85,B 0,C 180,E1 19393.241,E2 19393.241} C_VEL
LIN {X 0,Y 262.321,Z 560.76,A -85,B 0,C 180,E1 19398.606,E2 19398.606} C_VEL
LIN {X 0,Y 239.15,Z 577.84,A -85,B 0,C 180,E1 19406.362,E2 19406.362} C_VEL
LIN {X 0,Y 224.729,Z 587.034,A -85,B 0,C 180,E1 19414.029,E2 19414.029} C_VEL
LIN {X 0,Y 214.362,Z 591.501,A -85,B 0,C 180,E1 19423.588,E2 19423.588} C_VEL
LIN {X 0,Y 210.054,Z 590.562,A -85,B 0,C 180,E1 19431.71,E2 19431.71} C_VEL
LIN {X 0,Y 208.337,Z 584.197,A -85,B 0,C 180,E1 19441.038,E2 19441.038} C_VEL
LIN {X 0,Y 208.883,Z 573.227,A -85,B 0,C 180,E1 19449.382,E2 19449.382} C_VEL
LIN {X 0,Y 210.997,Z 558.019,A -85,B 0,C 180,E1 19456.898,E2 19456.898} C_VEL
LIN {X 0,Y 208.954,Z 548.059,A -85,B 0,C 180,E1 19460.797,E2 19460.797} C_VEL
LIN {X 0,Y 207.415,Z 536.935,A -85,B 0,C 180,E1 19464.531,E2 19464.531} C_VEL
LIN {X 0,Y 213.706,Z 508.928,A -85,B 0,C 180,E1 19471.386,E2 19471.386} C_VEL
LIN {X 0,Y 226.662,Z 503.876,A -85,B 0,C 180,E1 19475.681,E2 19475.681} C_VEL
LIN {X 0,Y 247.391,Z 493.848,A -85,B 0,C 180,E1 19479.979,E2 19479.979} C_VEL
LIN {X 0,Y 256.361,Z 488.991,A -85,B 0,C 180,E1 19481.452,E2 19481.452} C_VEL
LIN {X 0,Y 257.025,Z 490.748,A -85,B 0,C 180,E1 19482.078,E2 19482.078} C_VEL
LIN {X 0,Y 244.195,Z 518.234,A -85,B 0,C 180,E1 19486.423,E2 19486.423} C_VEL
LIN {X 0,Y 230.373,Z 542.449,A -85,B 0,C 180,E1 19492.323,E2 19492.323} C_VEL
LIN {X 0,Y 217.779,Z 561.954,A -85,B 0,C 180,E1 19499.742,E2 19499.742} C_VEL
LIN {X 0,Y 208.011,Z 576.207,A -85,B 0,C 180,E1 19508.666,E2 19508.666} C_VEL
LIN {X 0,Y 203.046,Z 583.962,A -85,B 0,C 180,E1 19517.081,E2 19517.081} C_VEL
LIN {X 0,Y 200.723,Z 587.682,A -85,B 0,C 180,E1 19525.681,E2 19525.681} C_VEL
LIN {X 0,Y 200.744,Z 587.645,A -85,B 0,C 180,E1 19534.332,E2 19534.332} C_VEL
LIN {X 0,Y 203.105,Z 583.852,A -85,B 0,C 180,E1 19542.928,E2 19542.928} C_VEL
LIN {X 0,Y 208.957,Z 574.761,A -85,B 0,C 180,E1 19552.363,E2 19552.363} C_VEL
LIN {X 0,Y 219.255,Z 559.603,A -85,B 0,C 180,E1 19561.196,E2 19561.196} C_VEL
LIN {X 0,Y 231.468,Z 540.498,A -85,B 0,C 180,E1 19568.137,E2 19568.137} C_VEL
LIN {X 0,Y 245.406,Z 515.54,A -85,B 0,C 180,E1 19573.957,E2 19573.957} C_VEL
LIN {X 0,Y 257.015,Z 489.588,A -85,B 0,C 180,E1 19578.048,E2 19578.048} C_VEL
LIN {X 0,Y 254.47,Z 467.703,A -85,B 0,C 180,E1 19583.852,E2 19583.852} C_VEL
LIN {X 0,Y 249.637,Z 449.669,A -85,B 0,C 180,E1 19589.477,E2 19589.477} C_VEL
LIN {X 0,Y 242.9,Z 432.434,A -85,B 0,C 180,E1 19596.47,E2 19596.47} C_VEL
LIN {X 0,Y 237.236,Z 421.2,A -85,B 0,C 180,E1 19603.25,E2 19603.25} C_VEL
LIN {X 0,Y 234.767,Z 415.698,A -85,B 0,C 180,E1 19607.668,E2 19607.668} C_VEL
LIN {X 0,Y 232.594,Z 409.889,A -85,B 0,C 180,E1 19616.271,E2 19616.271} C_VEL
LIN {X 0,Y 232.828,Z 410.882,A -85,B 0,C 180,E1 19620.987,E2 19620.987} C_VEL
LIN {X 0,Y 235.942,Z 417.421,A -85,B 0,C 180,E1 19629,E2 19629} C_VEL
LIN {X 0,Y 239.925,Z 425.408,A -85,B 0,C 180,E1 19634.505,E2 19634.505} C_VEL
LIN {X 0,Y 246.487,Z 438.217,A -85,B 0,C 180,E1 19640.955,E2 19640.955} C_VEL
LIN {X 0,Y 254.348,Z 458.632,A -85,B 0,C 180,E1 19647.906,E2 19647.906} C_VEL
LIN {X 0,Y 259.645,Z 479.974,A -85,B 0,C 180,E1 19653.432,E2 19653.432} C_VEL
LIN {X 0,Y 260.788,Z 488.139,A -85,B 0,C 180,E1 19655.27,E2 19655.27} C_VEL
LIN {X 0,Y 247.777,Z 520.937,A -85,B 0,C 180,E1 19659.168,E2 19659.168} C_VEL
LIN {X 0,Y 233.494,Z 550.134,A -85,B 0,C 180,E1 19664.495,E2 19664.495} C_VEL
LIN {X 0,Y 220.395,Z 574.149,A -85,B 0,C 180,E1 19671.177,E2 19671.177} C_VEL
LIN {X 0,Y 209.452,Z 594.071,A -85,B 0,C 180,E1 19679.598,E2 19679.598} C_VEL
LIN {X 0,Y 202.483,Z 608.646,A -85,B 0,C 180,E1 19689.354,E2 19689.354} C_VEL
LIN {X 0,Y 200.359,Z 615.736,A -85,B 0,C 180,E1 19696.892,E2 19696.892} C_VEL
LIN {X 0,Y 199.888,Z 619.974,A -85,B 0,C 180,E1 19705.65,E2 19705.65} C_VEL
LIN {X 0,Y 200.163,Z 620.59,A -85,B 0,C 180,E1 19709.994,E2 19709.994} C_VEL
LIN {X 0,Y 199.959,Z 618.41,A -85,B 0,C 180,E1 19718.703,E2 19718.703} C_VEL
LIN {X 0,Y 203.258,Z 611.785,A -85,B 0,C 180,E1 19731.858,E2 19731.858} C_VEL
LIN {X 0,Y 213.9,Z 600.202,A -85,B 0,C 180,E1 19743.137,E2 19743.137} C_VEL
LIN {X 0,Y 237.638,Z 579.68,A -85,B 0,C 180,E1 19754.482,E2 19754.482} C_VEL
LIN {X 0,Y 252.813,Z 567.938,A -85,B 0,C 180,E1 19758.796,E2 19758.796} C_VEL
LIN {X 0,Y 231.131,Z 581.771,A -85,B 0,C 180,E1 19766.166,E2 19766.166} C_VEL
LIN {X 0,Y 215.146,Z 590.152,A -85,B 0,C 180,E1 19775.024,E2 19775.024} C_VEL
LIN {X 0,Y 206.842,Z 592.61,A -85,B 0,C 180,E1 19782.974,E2 19782.974} C_VEL
LIN {X 0,Y 201.561,Z 590.074,A -85,B 0,C 180,E1 19793.528,E2 19793.528} C_VEL
LIN {X 0,Y 200.364,Z 583.038,A -85,B 0,C 180,E1 19802.162,E2 19802.162} C_VEL
LIN {X 0,Y 201.218,Z 571.203,A -85,B 0,C 180,E1 19810.633,E2 19810.633} C_VEL
LIN {X 0,Y 203.965,Z 553.451,A -85,B 0,C 180,E1 19818.946,E2 19818.946} C_VEL
LIN {X 0,Y 207.415,Z 536.935,A -85,B 0,C 180,E1 19824.531,E2 19824.531} C_VEL
LIN {X 0,Y 205.268,Z 529.199,A -85,B 0,C 180,E1 19826.947,E2 19826.947} C_VEL
LIN {X 0,Y 203.241,Z 520.974,A -85,B 0,C 180,E1 19829.281,E2 19829.281} C_VEL
LIN {X 0,Y 204.557,Z 516.294,A -85,B 0,C 180,E1 19830.581,E2 19830.581} C_VEL
LIN {X 0,Y 225.487,Z 509.034,A -85,B 0,C 180,E1 19837.172,E2 19837.172} C_VEL
LIN {X 0,Y 248.596,Z 498.323,A -85,B 0,C 180,E1 19841.603,E2 19841.603} C_VEL
LIN {X 0,Y 235.451,Z 524.512,A -85,B 0,C 180,E1 19846.281,E2 19846.281} C_VEL
LIN {X 0,Y 221.148,Z 547.775,A -85,B 0,C 180,E1 19852.594,E2 19852.594} C_VEL
LIN {X 0,Y 208.776,Z 565.624,A -85,B 0,C 180,E1 19860.245,E2 19860.245} C_VEL
LIN {X 0,Y 199,Z 579.191,A -85,B 0,C 180,E1 19869.987,E2 19869.987} C_VEL
LIN {X 0,Y 193.908,Z 586.962,A -85,B 0,C 180,E1 19881.023,E2 19881.023} C_VEL
LIN {X 0,Y 192.741,Z 588.8,A -85,B 0,C 180,E1 19890.007,E2 19890.007} C_VEL
LIN {X 0,Y 194.576,Z 585.804,A -85,B 0,C 180,E1 19901.223,E2 19901.223} C_VEL
LIN {X 0,Y 199.899,Z 577.938,A -85,B 0,C 180,E1 19911.091,E2 19911.091} C_VEL
LIN {X 0,Y 209.732,Z 564.207,A -85,B 0,C 180,E1 19920.358,E2 19920.358} C_VEL
LIN {X 0,Y 222.884,Z 544.907,A -85,B 0,C 180,E1 19928.236,E2 19928.236} C_VEL
LIN {X 0,Y 236.655,Z 522.128,A -85,B 0,C 180,E1 19934.09,E2 19934.09} C_VEL
LIN {X 0,Y 250.378,Z 494.658,A -85,B 0,C 180,E1 19938.716,E2 19938.716} C_VEL
LIN {X 0,Y 250.915,Z 486.916,A -85,B 0,C 180,E1 19940.574,E2 19940.574} C_VEL
LIN {X 0,Y 248.07,Z 465.682,A -85,B 0,C 180,E1 19946.687,E2 19946.687} C_VEL
LIN {X 0,Y 242.507,Z 446.694,A -85,B 0,C 180,E1 19953.602,E2 19953.602} C_VEL
LIN {X 0,Y 237.018,Z 433.369,A -85,B 0,C 180,E1 19960.41,E2 19960.41} C_VEL
LIN {X 0,Y 232.852,Z 423.356,A -85,B 0,C 180,E1 19967.756,E2 19967.756} C_VEL
LIN {X 0,Y 231.01,Z 417.817,A -85,B 0,C 180,E1 19976.245,E2 19976.245} C_VEL
LIN {X 0,Y 231.223,Z 418.892,A -85,B 0,C 180,E1 19981.063,E2 19981.063} C_VEL
LIN {X 0,Y 233.85,Z 425.05,A -85,B 0,C 180,E1 19988.671,E2 19988.671} C_VEL
LIN {X 0,Y 237.482,Z 432.897,A -85,B 0,C 180,E1 19994.186,E2 19994.186} C_VEL
LIN {X 0,Y 243.254,Z 445.385,A -85,B 0,C 180,E1 20000.543,E2 20000.543} C_VEL
LIN {X 0,Y 250.126,Z 465.291,A -85,B 0,C 180,E1 20007.487,E2 20007.487} C_VEL
LIN {X 0,Y 254.337,Z 485.546,A -85,B 0,C 180,E1 20012.889,E2 20012.889} C_VEL
LIN {X 0,Y 254.745,Z 491.599,A -85,B 0,C 180,E1 20014.259,E2 20014.259} C_VEL
LIN {X 0,Y 241.012,Z 523.893,A -85,B 0,C 180,E1 20018.253,E2 20018.253} C_VEL
LIN {X 0,Y 226.55,Z 551.767,A -85,B 0,C 180,E1 20023.587,E2 20023.587} C_VEL
LIN {X 0,Y 212.307,Z 576.592,A -85,B 0,C 180,E1 20030.92,E2 20030.92} C_VEL
LIN {X 0,Y 201.138,Z 595.706,A -85,B 0,C 180,E1 20039.762,E2 20039.762} C_VEL
LIN {X 0,Y 194.172,Z 609.984,A -85,B 0,C 180,E1 20050.34,E2 20050.34} C_VEL
LIN {X 0,Y 192.09,Z 617.74,A -85,B 0,C 180,E1 20060.924,E2 20060.924} C_VEL
LIN {X 0,Y 192.275,Z 619.951,A -85,B 0,C 180,E1 20069.993,E2 20069.993} C_VEL
LIN {X 0,Y 192.089,Z 617.765,A -85,B 0,C 180,E1 20079.062,E2 20079.062} C_VEL
LIN {X 0,Y 195.761,Z 611.664,A -85,B 0,C 180,E1 20092.741,E2 20092.741} C_VEL
LIN {X 0,Y 208.901,Z 599.557,A -85,B 0,C 180,E1 20105.427,E2 20105.427} C_VEL
LIN {X 0,Y 234.703,Z 580.25,A -85,B 0,C 180,E1 20116.517,E2 20116.517} C_VEL
LIN {X 0,Y 242.18,Z 575.081,A -85,B 0,C 180,E1 20118.595,E2 20118.595} C_VEL
LIN {X 0,Y 240.593,Z 575.915,A -85,B 0,C 180,E1 20119.646,E2 20119.646} C_VEL
LIN {X 0,Y 221.206,Z 586.255,A -85,B 0,C 180,E1 20126.801,E2 20126.801} C_VEL
LIN {X 0,Y 208.16,Z 591.763,A -85,B 0,C 180,E1 20134.125,E2 20134.125} C_VEL
LIN {X 0,Y 199.348,Z 593.59,A -85,B 0,C 180,E1 20142.313,E2 20142.313} C_VEL
LIN {X 0,Y 194.441,Z 591.534,A -85,B 0,C 180,E1 20151.039,E2 20151.039} C_VEL
LIN {X 0,Y 192.632,Z 585.223,A -85,B 0,C 180,E1 20159.997,E2 20159.997} C_VEL
LIN {X 0,Y 193.029,Z 573.841,A -85,B 0,C 180,E1 20169.022,E2 20169.022} C_VEL
LIN {X 0,Y 195.34,Z 557.593,A -85,B 0,C 180,E1 20177.474,E2 20177.474} C_VEL
LIN {X 0,Y 199.933,Z 535.514,A -85,B 0,C 180,E1 20185.357,E2 20185.357} C_VEL
LIN {X 0,Y 203.241,Z 520.974,A -85,B 0,C 180,E1 20189.281,E2 20189.281} C_VEL
LIN {X 0,Y 205.905,Z 516.952,A -85,B 0,C 180,E1 20191.179,E2 20191.179} C_VEL
LIN {X 0,Y 218.698,Z 516.238,A -85,B 0,C 180,E1 20197.375,E2 20197.375} C_VEL
LIN {X 0,Y 219.49,Z 515.985,A -85,B 0,C 180,E1 20197.586,E2 20197.586} C_VEL
LIN {X 0,Y 238.381,Z 508.35,A -85,B 0,C 180,E1 20201.492,E2 20201.492} C_VEL
LIN {X 0,Y 235.396,Z 515.305,A -85,B 0,C 180,E1 20202.927,E2 20202.927} C_VEL
LIN {X 0,Y 220.288,Z 540.581,A -85,B 0,C 180,E1 20208.802,E2 20208.802} C_VEL
LIN {X 0,Y 206.521,Z 560.165,A -85,B 0,C 180,E1 20216.024,E2 20216.024} C_VEL
LIN {X 0,Y 195.339,Z 574.894,A -85,B 0,C 180,E1 20224.777,E2 20224.777} C_VEL
LIN {X 0,Y 188.167,Z 584.533,A -85,B 0,C 180,E1 20234.887,E2 20234.887} C_VEL
LIN {X 0,Y 185.011,Z 588.956,A -85,B 0,C 180,E1 20245.313,E2 20245.313} C_VEL
LIN {X 0,Y 185.034,Z 588.921,A -85,B 0,C 180,E1 20254.7,E2 20254.7} C_VEL
LIN {X 0,Y 187.721,Z 585.135,A -85,B 0,C 180,E1 20264.008,E2 20264.008} C_VEL
LIN {X 0,Y 194.411,Z 576.049,A -85,B 0,C 180,E1 20274.139,E2 20274.139} C_VEL
LIN {X 0,Y 205.869,Z 560.919,A -85,B 0,C 180,E1 20283.48,E2 20283.48} C_VEL
LIN {X 0,Y 219.552,Z 541.437,A -85,B 0,C 180,E1 20290.811,E2 20290.811} C_VEL
LIN {X 0,Y 234.854,Z 515.977,A -85,B 0,C 180,E1 20296.829,E2 20296.829} C_VEL
LIN {X 0,Y 245.167,Z 495.079,A -85,B 0,C 180,E1 20300.231,E2 20300.231} C_VEL
LIN {X 0,Y 243.605,Z 473.773,A -85,B 0,C 180,E1 20306.53,E2 20306.53} C_VEL
LIN {X 0,Y 239.371,Z 455.419,A -85,B 0,C 180,E1 20313.219,E2 20313.219} C_VEL
LIN {X 0,Y 234.537,Z 441.344,A -85,B 0,C 180,E1 20320.194,E2 20320.194} C_VEL
LIN {X 0,Y 230.421,Z 430.691,A -85,B 0,C 180,E1 20328.383,E2 20328.383} C_VEL
LIN {X 0,Y 229.138,Z 425.63,A -85,B 0,C 180,E1 20336.214,E2 20336.214} C_VEL
LIN {X 0,Y 229.327,Z 426.771,A -85,B 0,C 180,E1 20341.072,E2 20341.072} C_VEL
LIN {X 0,Y 231.584,Z 432.574,A -85,B 0,C 180,E1 20348.368,E2 20348.368} C_VEL
LIN {X 0,Y 235.647,Z 441.763,A -85,B 0,C 180,E1 20354.893,E2 20354.893} C_VEL
LIN {X 0,Y 241.497,Z 457.315,A -85,B 0,C 180,E1 20362.097,E2 20362.097} C_VEL
LIN {X 0,Y 246.663,Z 476.33,A -85,B 0,C 180,E1 20368.405,E2 20368.405} C_VEL
LIN {X 0,Y 248.954,Z 494.205,A -85,B 0,C 180,E1 20373.071,E2 20373.071} C_VEL
LIN {X 0,Y 234.873,Z 525.481,A -85,B 0,C 180,E1 20377.084,E2 20377.084} C_VEL
LIN {X 0,Y 219.282,Z 554.101,A -85,B 0,C 180,E1 20382.793,E2 20382.793} C_VEL
LIN {X 0,Y 205.205,Z 577.162,A -85,B 0,C 180,E1 20389.982,E2 20389.982} C_VEL
LIN {X 0,Y 194.145,Z 594.964,A -85,B 0,C 180,E1 20398.505,E2 20398.505} C_VEL
LIN {X 0,Y 186.54,Z 609.322,A -85,B 0,C 180,E1 20409.501,E2 20409.501} C_VEL
LIN {X 0,Y 184.238,Z 617.096,A -85,B 0,C 180,E1 20420.534,E2 20420.534} C_VEL
LIN {X 0,Y 184.388,Z 619.313,A -85,B 0,C 180,E1 20429.993,E2 20429.993} C_VEL
LIN {X 0,Y 184.238,Z 617.078,A -85,B 0,C 180,E1 20439.561,E2 20439.561} C_VEL
LIN {X 0,Y 189.946,Z 610.03,A -85,B 0,C 180,E1 20455.992,E2 20455.992} C_VEL
LIN {X 0,Y 205.93,Z 597.975,A -85,B 0,C 180,E1 20468.666,E2 20468.666} C_VEL
LIN {X 0,Y 232.966,Z 580.486,A -85,B 0,C 180,E1 20478.808,E2 20478.808} C_VEL
LIN {X 0,Y 227.631,Z 582.98,A -85,B 0,C 180,E1 20480.813,E2 20480.813} C_VEL
LIN {X 0,Y 207.621,Z 591.408,A -85,B 0,C 180,E1 20489.305,E2 20489.305} C_VEL
LIN {X 0,Y 193.091,Z 594.607,A -85,B 0,C 180,E1 20500.176,E2 20500.176} C_VEL
LIN {X 0,Y 186.635,Z 591.968,A -85,B 0,C 180,E1 20510.66,E2 20510.66} C_VEL
LIN {X 0,Y 184.622,Z 583.868,A -85,B 0,C 180,E1 20521.172,E2 20521.172} C_VEL
LIN {X 0,Y 185.433,Z 571.153,A -85,B 0,C 180,E1 20530.65,E2 20530.65} C_VEL
LIN {X 0,Y 188.238,Z 553.513,A -85,B 0,C 180,E1 20539.372,E2 20539.372} C_VEL
LIN {X 0,Y 193.654,Z 529.287,A -85,B 0,C 180,E1 20547.584,E2 20547.584} C_VEL
LIN {X 0,Y 195.135,Z 523.667,A -85,B 0,C 180,E1 20549.32,E2 20549.32} C_VEL
LIN {X 0,Y 205.559,Z 520.68,A -85,B 0,C 180,E1 20553.526,E2 20553.526} C_VEL
LIN {X 0,Y 219.49,Z 515.985,A -85,B 0,C 180,E1 20557.586,E2 20557.586} C_VEL
LIN {X 0,Y 223.524,Z 516.737,A -85,B 0,C 180,E1 20559.46,E2 20559.46} C_VEL
LIN {X 0,Y 227.833,Z 517.381,A -85,B 0,C 180,E1 20561.24,E2 20561.24} C_VEL
LIN {X 0,Y 228.775,Z 517.042,A -85,B 0,C 180,E1 20561.43,E2 20561.43} C_VEL
LIN {X 0,Y 227.228,Z 521.048,A -85,B 0,C 180,E1 20562.454,E2 20562.454} C_VEL
LIN {X 0,Y 212.177,Z 544.402,A -85,B 0,C 180,E1 20568.395,E2 20568.395} C_VEL
LIN {X 0,Y 197.631,Z 563.899,A -85,B 0,C 180,E1 20576.271,E2 20576.271} C_VEL
LIN {X 0,Y 186.078,Z 578.137,A -85,B 0,C 180,E1 20586.004,E2 20586.004} C_VEL
LIN {X 0,Y 180.019,Z 585.88,A -85,B 0,C 180,E1 20595.394,E2 20595.394} C_VEL
LIN {X 0,Y 177.183,Z 589.592,A -85,B 0,C 180,E1 20605.106,E2 20605.106} C_VEL
LIN {X 0,Y 177.206,Z 589.556,A -85,B 0,C 180,E1 20614.908,E2 20614.908} C_VEL
LIN {X 0,Y 180.641,Z 585.013,A -85,B 0,C 180,E1 20625.87,E2 20625.87} C_VEL
LIN {X 0,Y 188.316,Z 575.34,A -85,B 0,C 180,E1 20636.25,E2 20636.25} C_VEL
LIN {X 0,Y 200.947,Z 559.488,A -85,B 0,C 180,E1 20645.732,E2 20645.732} C_VEL
LIN {X 0,Y 215.903,Z 538.748,A -85,B 0,C 180,E1 20653.175,E2 20653.175} C_VEL
LIN {X 0,Y 231.48,Z 513.297,A -85,B 0,C 180,E1 20658.895,E2 20658.895} C_VEL
LIN {X 0,Y 239.231,Z 498.403,A -85,B 0,C 180,E1 20661.227,E2 20661.227} C_VEL
LIN {X 0,Y 238.538,Z 478.921,A -85,B 0,C 180,E1 20667.279,E2 20667.279} C_VEL
LIN {X 0,Y 234.864,Z 460.172,A -85,B 0,C 180,E1 20674.493,E2 20674.493} C_VEL
LIN {X 0,Y 231.187,Z 447.976,A -85,B 0,C 180,E1 20680.89,E2 20680.89} C_VEL
LIN {X 0,Y 228.042,Z 438.198,A -85,B 0,C 180,E1 20688.515,E2 20688.515} C_VEL
LIN {X 0,Y 226.964,Z 433.417,A -85,B 0,C 180,E1 20696.178,E2 20696.178} C_VEL
LIN {X 0,Y 227.119,Z 434.393,A -85,B 0,C 180,E1 20700.861,E2 20700.861} C_VEL
LIN {X 0,Y 228.964,Z 439.43,A -85,B 0,C 180,E1 20707.602,E2 20707.602} C_VEL
LIN {X 0,Y 232.503,Z 448.715,A -85,B 0,C 180,E1 20714.376,E2 20714.376} C_VEL
LIN {X 0,Y 237.53,Z 463.672,A -85,B 0,C 180,E1 20721.501,E2 20721.501} C_VEL
LIN {X 0,Y 241.887,Z 482.692,A -85,B 0,C 180,E1 20728,E2 20728} C_VEL
LIN {X 0,Y 243.375,Z 495.997,A -85,B 0,C 180,E1 20731.723,E2 20731.723} C_VEL
LIN {X 0,Y 228.85,Z 527.071,A -85,B 0,C 180,E1 20735.857,E2 20735.857} C_VEL
LIN {X 0,Y 212.744,Z 555.137,A -85,B 0,C 180,E1 20741.642,E2 20741.642} C_VEL
LIN {X 0,Y 197.829,Z 578.245,A -85,B 0,C 180,E1 20749.187,E2 20749.187} C_VEL
LIN {X 0,Y 186.157,Z 596.02,A -85,B 0,C 180,E1 20758.275,E2 20758.275} C_VEL
LIN {X 0,Y 178.995,Z 608.57,A -85,B 0,C 180,E1 20768.5,E2 20768.5} C_VEL
LIN {X 0,Y 176.351,Z 616.449,A -85,B 0,C 180,E1 20780.106,E2 20780.106} C_VEL
LIN {X 0,Y 176.529,Z 618.677,A -85,B 0,C 180,E1 20789.993,E2 20789.993} C_VEL
LIN {X 0,Y 176.372,Z 616.477,A -85,B 0,C 180,E1 20799.878,E2 20799.878} C_VEL
LIN {X 0,Y 182.698,Z 609.861,A -85,B 0,C 180,E1 20817.106,E2 20817.106} C_VEL
LIN {X 0,Y 199.821,Z 598.92,A -85,B 0,C 180,E1 20830.082,E2 20830.082} C_VEL
LIN {X 0,Y 221.997,Z 586.2,A -85,B 0,C 180,E1 20838.595,E2 20838.595} C_VEL
LIN {X 0,Y 223.073,Z 585.521,A -85,B 0,C 180,E1 20839.287,E2 20839.287} C_VEL
LIN {X 0,Y 201.072,Z 593.321,A -85,B 0,C 180,E1 20848.191,E2 20848.191} C_VEL
LIN {X 0,Y 188.785,Z 595.625,A -85,B 0,C 180,E1 20856.359,E2 20856.359} C_VEL
LIN {X 0,Y 179.824,Z 593.402,A -85,B 0,C 180,E1 20867.847,E2 20867.847} C_VEL
LIN {X 0,Y 176.978,Z 586.032,A -85,B 0,C 180,E1 20878.771,E2 20878.771} C_VEL
LIN {X 0,Y 177.176,Z 574.226,A -85,B 0,C 180,E1 20888.597,E2 20888.597} C_VEL
LIN {X 0,Y 179.579,Z 557.501,A -85,B 0,C 180,E1 20897.791,E2 20897.791} C_VEL
LIN {X 0,Y 184.296,Z 535.859,A -85,B 0,C 180,E1 20906.045,E2 20906.045} C_VEL
LIN {X 0,Y 185.722,Z 530.436,A -85,B 0,C 180,E1 20907.833,E2 20907.833} C_VEL
LIN {X 0,Y 191.483,Z 529.361,A -85,B 0,C 180,E1 20910.921,E2 20910.921} C_VEL
LIN {X 0,Y 218.876,Z 520.779,A -85,B 0,C 180,E1 20919.382,E2 20919.382} C_VEL
LIN {X 0,Y 227.833,Z 517.381,A -85,B 0,C 180,E1 20921.24,E2 20921.24} C_VEL
LIN {X 0,Y 227.331,Z 519.877,A -85,B 0,C 180,E1 20922.018,E2 20922.018} C_VEL
LIN {X 0,Y 215.074,Z 532.755,A -85,B 0,C 180,E1 20923.479,E2 20923.479} C_VEL
LIN {X 0,Y 214.114,Z 534.057,A -85,B 0,C 180,E1 20923.773,E2 20923.773} C_VEL
LIN {X 0,Y 198.005,Z 555.94,A -85,B 0,C 180,E1 20930.9,E2 20930.9} C_VEL
LIN {X 0,Y 184.874,Z 571.879,A -85,B 0,C 180,E1 20939.409,E2 20939.409} C_VEL
LIN {X 0,Y 175.181,Z 583.199,A -85,B 0,C 180,E1 20949.784,E2 20949.784} C_VEL
LIN {X 0,Y 170.588,Z 588.872,A -85,B 0,C 180,E1 20959.784,E2 20959.784} C_VEL
LIN {X 0,Y 169.112,Z 590.711,A -85,B 0,C 180,E1 20970.008,E2 20970.008} C_VEL
LIN {X 0,Y 171.292,Z 587.839,A -85,B 0,C 180,E1 20982.506,E2 20982.506} C_VEL
LIN {X 0,Y 177.937,Z 579.873,A -85,B 0,C 180,E1 20993.845,E2 20993.845} C_VEL
LIN {X 0,Y 189.613,Z 566.167,A -85,B 0,C 180,E1 21003.988,E2 21003.988} C_VEL
LIN {X 0,Y 204.944,Z 546.78,A -85,B 0,C 180,E1 21012.384,E2 21012.384} C_VEL
LIN {X 0,Y 220.283,Z 524.259,A -85,B 0,C 180,E1 21018.375,E2 21018.375} C_VEL
LIN {X 0,Y 233.46,Z 500.663,A -85,B 0,C 180,E1 21022.574,E2 21022.574} C_VEL
LIN {X 0,Y 233.115,Z 481.008,A -85,B 0,C 180,E1 21029.12,E2 21029.12} C_VEL
LIN {X 0,Y 230.217,Z 463.986,A -85,B 0,C 180,E1 21036.25,E2 21036.25} C_VEL
LIN {X 0,Y 226.808,Z 451.436,A -85,B 0,C 180,E1 21043.763,E2 21043.763} C_VEL
LIN {X 0,Y 225.45,Z 446.005,A -85,B 0,C 180,E1 21048.381,E2 21048.381} C_VEL
LIN {X 0,Y 224.55,Z 441.138,A -85,B 0,C 180,E1 21056.137,E2 21056.137} C_VEL
LIN {X 0,Y 224.778,Z 441.26,A -85,B 0,C 180,E1 21060.003,E2 21060.003} C_VEL
LIN {X 0,Y 226.326,Z 447.296,A -85,B 0,C 180,E1 21067.691,E2 21067.691} C_VEL
LIN {X 0,Y 229.413,Z 456.407,A -85,B 0,C 180,E1 21074.33,E2 21074.33} C_VEL
LIN {X 0,Y 233.657,Z 471.136,A -85,B 0,C 180,E1 21081.377,E2 21081.377} C_VEL
LIN {X 0,Y 236.997,Z 489.793,A -85,B 0,C 180,E1 21087.87,E2 21087.87} C_VEL
LIN {X 0,Y 237.282,Z 499.925,A -85,B 0,C 180,E1 21090.647,E2 21090.647} C_VEL
LIN {X 0,Y 221.688,Z 530.914,A -85,B 0,C 180,E1 21094.956,E2 21094.956} C_VEL
LIN {X 0,Y 205.256,Z 557.752,A -85,B 0,C 180,E1 21100.876,E2 21100.876} C_VEL
LIN {X 0,Y 190.198,Z 579.728,A -85,B 0,C 180,E1 21108.495,E2 21108.495} C_VEL
LIN {X 0,Y 177.908,Z 597.401,A -85,B 0,C 180,E1 21118.321,E2 21118.321} C_VEL
LIN {X 0,Y 170.72,Z 609.345,A -85,B 0,C 180,E1 21129.216,E2 21129.216} C_VEL
LIN {X 0,Y 168.476,Z 615.801,A -85,B 0,C 180,E1 21139.639,E2 21139.639} C_VEL
LIN {X 0,Y 168.637,Z 618.039,A -85,B 0,C 180,E1 21149.992,E2 21149.992} C_VEL
LIN {X 0,Y 168.519,Z 615.832,A -85,B 0,C 180,E1 21160.343,E2 21160.343} C_VEL
LIN {X 0,Y 169.202,Z 613.37,A -85,B 0,C 180,E1 21165.563,E2 21165.563} C_VEL
LIN {X 0,Y 177.791,Z 608.366,A -85,B 0,C 180,E1 21180.716,E2 21180.716} C_VEL
LIN {X 0,Y 197.989,Z 597.639,A -85,B 0,C 180,E1 21193.478,E2 21193.478} C_VEL
LIN {X 0,Y 212.067,Z 590.524,A -85,B 0,C 180,E1 21198.677,E2 21198.677} C_VEL
LIN {X 0,Y 212.783,Z 590.009,A -85,B 0,C 180,E1 21199.517,E2 21199.517} C_VEL
LIN {X 0,Y 194.578,Z 595.113,A -85,B 0,C 180,E1 21206.997,E2 21206.997} C_VEL
LIN {X 0,Y 181.632,Z 596.73,A -85,B 0,C 180,E1 21215.367,E2 21215.367} C_VEL
LIN {X 0,Y 172.124,Z 593.797,A -85,B 0,C 180,E1 21227.294,E2 21227.294} C_VEL
LIN {X 0,Y 169.087,Z 585.734,A -85,B 0,C 180,E1 21238.714,E2 21238.714} C_VEL
LIN {X 0,Y 169.469,Z 572.428,A -85,B 0,C 180,E1 21249.639,E2 21249.639} C_VEL
LIN {X 0,Y 172.271,Z 554.636,A -85,B 0,C 180,E1 21259.238,E2 21259.238} C_VEL
LIN {X 0,Y 176.419,Z 536.94,A -85,B 0,C 180,E1 21266.32,E2 21266.32} C_VEL
LIN {X 0,Y 191.207,Z 533.564,A -85,B 0,C 180,E1 21273.654,E2 21273.654} C_VEL
LIN {X 0,Y 219.472,Z 524.823,A -85,B 0,C 180,E1 21281.396,E2 21281.396} C_VEL
LIN {X 0,Y 216.7,Z 530.157,A -85,B 0,C 180,E1 21282.823,E2 21282.823} C_VEL
LIN {X 0,Y 214.114,Z 534.057,A -85,B 0,C 180,E1 21283.773,E2 21283.773} C_VEL
LIN {X 0,Y 203.644,Z 545.307,A -85,B 0,C 180,E1 21286.104,E2 21286.104} C_VEL
LIN {X 0,Y 192.98,Z 555.356,A -85,B 0,C 180,E1 21288.886,E2 21288.886} C_VEL
LIN {X 0,Y 178.758,Z 571.779,A -85,B 0,C 180,E1 21297.599,E2 21297.599} C_VEL
LIN {X 0,Y 167.777,Z 583.839,A -85,B 0,C 180,E1 21308.85,E2 21308.85} C_VEL
LIN {X 0,Y 162.815,Z 589.511,A -85,B 0,C 180,E1 21319.29,E2 21319.29} C_VEL
LIN {X 0,Y 161.235,Z 591.349,A -85,B 0,C 180,E1 21330.008,E2 21330.008} C_VEL
LIN {X 0,Y 163.415,Z 588.695,A -85,B 0,C 180,E1 21342.595,E2 21342.595} C_VEL
LIN {X 0,Y 170.73,Z 580.517,A -85,B 0,C 180,E1 21354.919,E2 21354.919} C_VEL
LIN {X 0,Y 183.118,Z 566.816,A -85,B 0,C 180,E1 21365.37,E2 21365.37} C_VEL
